KUKA KRL program: MyProgram_084().src

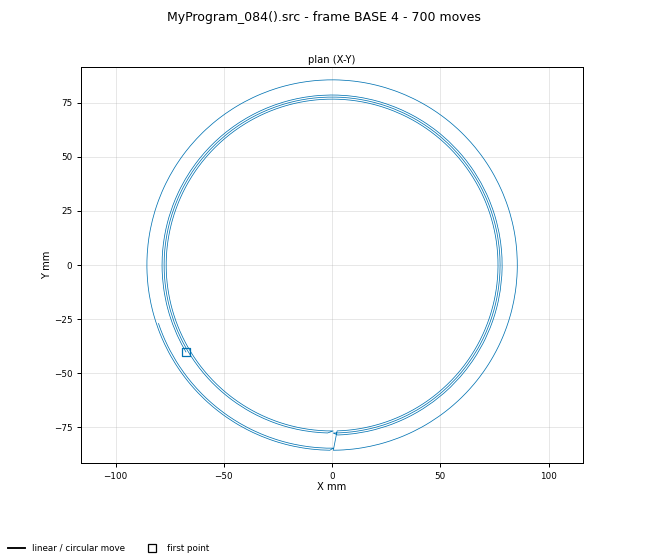
[picture p0: tool path of MyProgram_084().src in frame BASE 4, 700 of 700 moves have a stored position in this frame; points joined in program order, loops and branches not executed]
&ACCESS RVP
&REL 1
&PARAM TEMPLATE = C:\KRC\Roboter\Template\vorgabe
&PARAM EDITMASK = *
DEF MyProgram_084()
; ---- Setting reference (Base) ----
$BASE = BASE_DATA[4]

; --------------------------
; ---- Setting tool (TCP) ----
$TOOL = TOOL_DATA[3]
; --------------------------

$VEL.CP = VEL_APROX_PRINT
Startdeposition()
$VEL.CP = VEL_PRINT
LIN {X -67.4962,Y -40.1189,Z 83,A -155.1971,B 24.913,C -2.1538,E1 24.8612,E2 239.9035} C_DIS
LIN {X -69.3638,Y -36.7975,Z 83,A -157.7147,B 24.9119,C -2.1678,E1 24.8579,E2 242.401} C_DIS
LIN {X -71.5627,Y -32.3128,Z 83,A -161.7779,B 24.9119,C -2.1676,E1 24.853,E2 246.4869} C_DIS
LIN {X -73.6163,Y -27.3162,Z 83,A -165.4446,B 24.9104,C -2.1857,E1 24.8493,E2 250.1308} C_DIS
LIN {X -75.14,Y -22.7935,Z 83,A -168.9954,B 24.9097,C -2.1943,E1 24.8462,E2 253.6814} C_DIS
LIN {X -76.0413,Y -19.5719,Z 83,A -171.3695,B 24.9089,C -2.2034,E1 24.8445,E2 256.0476} C_DIS
LIN {X -76.5834,Y -17.3332,Z 83,A -173.4714,B 24.9094,C -2.1982,E1 24.8432,E2 258.1743} C_DIS
LIN {X -77.4433,Y -12.9563,Z 83,A -176.3604,B 24.9078,C -2.2172,E1 24.8417,E2 261.035} C_DIS
LIN {X -77.8334,Y -10.3623,Z 83,A -178.4896,B 24.9078,C -2.2179,E1 24.8409,E2 263.1752} C_DIS
LIN {X -78.3135,Y -5.7007,Z 83,A 178.2886,B 24.9064,C -2.2335,E1 24.8401,E2 266.3791} C_DIS
LIN {X -78.4754,Y -2.6451,Z 83,A 176.0932,B 24.9057,C -2.2415,E1 24.8398,E2 268.5686} C_DIS
LIN {X -78.5203,Y -0.1798,Z 83,A 174.0288,B 24.9058,C -2.2407,E1 24.8398,E2 270.6472} C_DIS
LIN {X -78.4321,Y 3.7214,Z 83,A 171.4381,B 24.9045,C -2.2561,E1 24.84,E2 273.217} C_DIS
LIN {X -78.2302,Y 6.7519,Z 83,A 169.0363,B 24.9043,C -2.2586,E1 24.8405,E2 275.6272} C_DIS
LIN {X -77.8931,Y 9.901,Z 83,A 166.9372,B 24.9032,C -2.2711,E1 24.8412,E2 277.7088} C_DIS
LIN {X -77.3929,Y 13.2579,Z 83,A 164.5258,B 24.9024,C -2.2806,E1 24.8423,E2 280.1121} C_DIS
LIN {X -76.7687,Y 16.4912,Z 83,A 161.8494,B 24.9024,C -2.2815,E1 24.8437,E2 282.8021} C_DIS
LIN {X -76.0396,Y 19.5784,Z 83,A 159.9359,B 24.9009,C -2.2986,E1 24.845,E2 284.6859} C_DIS
LIN {X -75.3479,Y 22.0927,Z 83,A 157.1821,B 24.9022,C -2.2837,E1 24.8471,E2 287.4912} C_DIS
LIN {X -73.5762,Y 27.4236,Z 83,A 153.3028,B 24.9006,C -2.3017,E1 24.8507,E2 291.3496} C_DIS
LIN {X -72.4018,Y 30.3864,Z 83,A 151.2241,B 24.8995,C -2.3147,E1 24.8529,E2 293.4087} C_DIS
LIN {X -70.9859,Y 33.5643,Z 83,A 148.6946,B 24.8988,C -2.3225,E1 24.8558,E2 295.9336} C_DIS
LIN {X -69.965,Y 35.6404,Z 83,A 146.6894,B 24.899,C -2.3197,E1 24.8583,E2 297.9562} C_DIS
LIN {X -67.7859,Y 39.6302,Z 83,A 143.1182,B 24.8988,C -2.323,E1 24.8633,E2 301.5383} C_DIS
LIN {X -65.3999,Y 43.4542,Z 83,A 139.7994,B 24.898,C -2.3314,E1 24.8683,E2 304.8537} C_DIS
LIN {X -63.0593,Y 46.7874,Z 83,A 137.4432,B 24.896,C -2.3546,E1 24.8721,E2 307.166} C_DIS
LIN {X -61.1985,Y 49.1953,Z 83,A 134.8431,B 24.8963,C -2.351,E1 24.8766,E2 309.7869} C_DIS
LIN {X -58.9466,Y 51.8721,Z 83,A 132.515,B 24.8952,C -2.3631,E1 24.8808,E2 312.0968} C_DIS
LIN {X -56.6359,Y 54.385,Z 83,A 129.9158,B 24.8949,C -2.3665,E1 24.8858,E2 314.6992} C_DIS
LIN {X -54.1507,Y 56.8608,Z 83,A 127.2895,B 24.8945,C -2.3708,E1 24.8911,E2 317.3261} C_DIS
LIN {X -51.3752,Y 59.3806,Z 83,A 124.709,B 24.8936,C -2.3809,E1 24.8964,E2 319.8928} C_DIS
LIN {X -48.7716,Y 61.536,Z 83,A 122.1128,B 24.8934,C -2.383,E1 24.9021,E2 322.4938} C_DIS
LIN {X -45.6856,Y 63.8605,Z 83,A 118.9561,B 24.8937,C -2.3802,E1 24.9092,E2 325.6683} C_DIS
LIN {X -42.8175,Y 65.8196,Z 83,A 115.9085,B 24.8944,C -2.372,E1 24.9164,E2 328.7453} C_DIS
LIN {X -39.3112,Y 67.9707,Z 83,A 113.6601,B 24.8922,C -2.3965,E1 24.9217,E2 330.9422} C_DIS
LIN {X -36.2205,Y 69.6677,Z 83,A 111.1741,B 24.8916,C -2.403,E1 24.9278,E2 333.4195} C_DIS
LIN {X -33.3372,Y 71.0916,Z 83,A 108.8468,B 24.8913,C -2.4072,E1 24.9336,E2 335.7429} C_DIS
LIN {X -30.2227,Y 72.4708,Z 83,A 105.584,B 24.8928,C -2.3906,E1 24.9422,E2 339.0527} C_DIS
LIN {X -26.6807,Y 73.848,Z 83,A 103.7974,B 24.8901,C -2.4199,E1 24.9467,E2 340.7734} C_DIS
LIN {X -22.5013,Y 75.2267,Z 83,A 100.3905,B 24.8902,C -2.4184,E1 24.9558,E2 344.1897} C_DIS
LIN {X -19.5528,Y 76.0462,Z 83,A 98.0831,B 24.8902,C -2.4187,E1 24.962,E2 346.5} C_DIS
LIN {X -16.2475,Y 76.8217,Z 83,A 95.2262,B 24.8909,C -2.4108,E1 24.9698,E2 349.3794} C_DIS
LIN {X -12.6748,Y 77.4904,Z 83,A 92.5015,B 24.8909,C -2.4108,E1 24.9773,E2 352.1066} C_DIS
LIN {X -8.3982,Y 78.0696,Z 83,A 89.8262,B 24.8896,C -2.4253,E1 24.9847,E2 354.7492} C_DIS
LIN {X -5.2916,Y 78.3411,Z 83,A 87.2441,B 24.8903,C -2.418,E1 24.9919,E2 357.3497} C_DIS
LIN {X -0.6851,Y 78.5169,Z 83,A 84.1569,B 24.8895,C -2.4265,E1 25.0005,E2 360.4172} C_DIS
LIN {X 2.6698,Y 78.4747,Z 83,A 81.8017,B 24.8892,C -2.4293,E1 25.007,E2 362.7652} C_DIS
LIN {X 7.1476,Y 78.1937,Z 83,A 78.4133,B 24.8895,C -2.4261,E1 25.0165,E2 366.1598} C_DIS
LIN {X 10.8186,Y 77.7711,Z 83,A 75.7639,B 24.8895,C -2.4268,E1 25.0238,E2 368.8054} C_DIS
LIN {X 14.4011,Y 77.189,Z 83,A 72.6133,B 24.8908,C -2.4119,E1 25.0326,E2 371.9879} C_DIS
LIN {X 18.7763,Y 76.2418,Z 83,A 69.7445,B 24.89,C -2.4213,E1 25.0403,E2 374.8305} C_DIS
LIN {X 21.894,Y 75.4069,Z 83,A 67.3804,B 24.8901,C -2.4194,E1 25.0466,E2 377.195} C_DIS
LIN {X 25.0356,Y 74.4215,Z 83,A 65.1631,B 24.8898,C -2.4228,E1 25.0525,E2 379.4002} C_DIS
LIN {X 29.0768,Y 72.9386,Z 83,A 62.2037,B 24.8896,C -2.4251,E1 25.0602,E2 382.348} C_DIS
LIN {X 32.2098,Y 71.6091,Z 83,A 59.24,B 24.8911,C -2.4086,E1 25.0679,E2 385.3435} C_DIS
LIN {X 35.5962,Y 69.9876,Z 83,A 56.777,B 24.8907,C -2.4132,E1 25.074,E2 387.7891} C_DIS
LIN {X 38.5611,Y 68.3994,Z 83,A 53.5616,B 24.893,C -2.3878,E1 25.082,E2 391.0551} C_DIS
LIN {X 41.7678,Y 66.4893,Z 83,A 51.5388,B 24.8915,C -2.404,E1 25.0867,E2 393.0331} C_DIS
LIN {X 43.7872,Y 65.1774,Z 83,A 49.4601,B 24.8926,C -2.3918,E1 25.0915,E2 395.1338} C_DIS
LIN {X 47.0859,Y 62.8352,Z 83,A 46.9103,B 24.892,C -2.3985,E1 25.0972,E2 397.6586} C_DIS
LIN {X 49.6786,Y 60.8068,Z 83,A 44.6975,B 24.892,C -2.3998,E1 25.102,E2 399.8603} C_DIS
LIN {X 53.8865,Y 57.1104,Z 83,A 40.3742,B 24.8933,C -2.3847,E1 25.1111,E2 404.202} C_DIS
LIN {X 58.1887,Y 52.722,Z 83,A 35.9551,B 24.894,C -2.3769,E1 25.1196,E2 408.6203} C_DIS
LIN {X 60.2405,Y 50.3634,Z 83,A 33.7323,B 24.8943,C -2.3735,E1 25.1237,E2 410.8412} C_DIS
LIN {X 62.2799,Y 47.818,Z 83,A 30.7906,B 24.8963,C -2.3509,E1 25.1288,E2 413.8223} C_DIS
LIN {X 64.1977,Y 45.2131,Z 83,A 28.9176,B 24.8955,C -2.3597,E1 25.1318,E2 415.6654} C_DIS
LIN {X 65.697,Y 43.0036,Z 83,A 26.6513,B 24.8968,C -2.3452,E1 25.1353,E2 417.9548} C_DIS
LIN {X 68.7357,Y 37.9588,Z 83,A 23.018,B 24.896,C -2.354,E1 25.1404,E2 421.5486} C_DIS
LIN {X 71.3889,Y 32.6985,Z 83,A 18.4593,B 24.8978,C -2.3341,E1 25.146,E2 426.1299} C_DIS
LIN {X 72.7,Y 29.6657,Z 83,A 15.8312,B 24.899,C -2.3206,E1 25.1489,E2 428.7754} C_DIS
LIN {X 74.1369,Y 25.8663,Z 83,A 13.2522,B 24.8987,C -2.3238,E1 25.1513,E2 431.3324} C_DIS
LIN {X 75.1174,Y 22.8665,Z 83,A 11.1082,B 24.8989,C -2.3218,E1 25.1531,E2 433.4689} C_DIS
LIN {X 75.9431,Y 19.954,Z 83,A 8.9268,B 24.8994,C -2.316,E1 25.1548,E2 435.6515} C_DIS
LIN {X 77.1297,Y 14.7088,Z 83,A 4.8617,B 24.9008,C -2.2996,E1 25.1572,E2 439.7318} C_DIS
LIN {X 77.7907,Y 10.6646,Z 83,A 1.7462,B 24.9019,C -2.2864,E1 25.1585,E2 442.8601} C_DIS
LIN {X 78.2253,Y 6.7842,Z 83,A -1.4293,B 24.9036,C -2.2673,E1 25.1594,E2 446.0619} C_DIS
LIN {X 78.4503,Y 3.3007,Z 83,A -4.5335,B 24.9057,C -2.2421,E1 25.1598,E2 449.2071} C_DIS
LIN {X 78.5112,Y -1.1833,Z 83,A -6.7555,B 24.9038,C -2.2641,E1 25.1598,E2 451.364} C_DIS
LIN {X 78.3698,Y -4.8681,Z 83,A -9.4916,B 24.9047,C -2.2541,E1 25.1594,E2 454.1076} C_DIS
LIN {X 77.6444,Y -11.6949,Z 83,A -14.1193,B 24.905,C -2.25,E1 25.1579,E2 458.7174} C_DIS
LIN {X 76.7025,Y -16.7949,Z 83,A -18.2468,B 24.9069,C -2.2273,E1 25.1558,E2 462.8745} C_DIS
LIN {X 76.0708,Y -19.4568,Z 83,A -20.7555,B 24.9088,C -2.2051,E1 25.154,E2 465.421} C_DIS
LIN {X 75.1954,Y -22.607,Z 83,A -22.6705,B 24.9082,C -2.2123,E1 25.1525,E2 467.3083} C_DIS
LIN {X 74.1573,Y -25.8085,Z 83,A -24.9152,B 24.9082,C -2.2112,E1 25.1505,E2 469.5427} C_DIS
LIN {X 73.0003,Y -28.9196,Z 83,A -27.6923,B 24.9098,C -2.1928,E1 25.1477,E2 472.3479} C_DIS
LIN {X 70.715,Y -34.1282,Z 83,A -31.553,B 24.9101,C -2.1894,E1 25.1433,E2 476.1958} C_DIS
LIN {X 69.6417,Y -36.2699,Z 83,A -33.8227,B 24.9118,C -2.1682,E1 25.1403,E2 478.5035} C_DIS
LIN {X 66.7563,Y -41.3403,Z 83,A -37.3323,B 24.9109,C -2.179,E1 25.1354,E2 481.9695} C_DIS
LIN {X 64.7944,Y -44.3529,Z 83,A -39.7414,B 24.9109,C -2.1783,E1 25.1317,E2 484.3682} C_DIS
LIN {X 62.0109,Y -48.1672,Z 83,A -43.4052,B 24.9123,C -2.1623,E1 25.1256,E2 488.0523} C_DIS
LIN {X 59.1059,Y -51.6897,Z 83,A -46.8855,B 24.9134,C -2.1491,E1 25.1193,E2 491.5478} C_DIS
LIN {X 54.589,Y -56.4393,Z 83,A -51.2634,B 24.9134,C -2.1497,E1 25.1109,E2 495.9053} C_DIS
LIN {X 51.7179,Y -59.0813,Z 83,A -54.4123,B 24.9146,C -2.134,E1 25.1043,E2 499.0789} C_DIS
LIN {X 46.8486,Y -63.0135,Z 83,A -59.0188,B 24.9155,C -2.1229,E1 25.0942,E2 503.6943} C_DIS
LIN {X 41.9662,Y -66.3653,Z 83,A -63.0379,B 24.9155,C -2.1235,E1 25.085,E2 507.6986} C_DIS
LIN {X 39.4629,Y -67.8835,Z 83,A -65.1401,B 24.9157,C -2.1206,E1 25.0799,E2 509.8011} C_DIS
LIN {X 36.5498,Y -69.4942,Z 83,A -68.3691,B 24.9179,C -2.0927,E1 25.0718,E2 513.087} C_DIS
LIN {X 33.6867,Y -70.9272,Z 83,A -70.1646,B 24.9169,C -2.1049,E1 25.0674,E2 514.8488} C_DIS
LIN {X 31.1101,Y -72.0942,Z 83,A -72.9633,B 24.9188,C -2.0803,E1 25.0601,E2 517.699} C_DIS
LIN {X 27.621,Y -73.5014,Z 83,A -74.9496,B 24.9174,C -2.0987,E1 25.055,E2 519.6373} C_DIS
LIN {X 24.8884,Y -74.4711,Z 83,A -76.8881,B 24.9172,C -2.1013,E1 25.0499,E2 521.566} C_DIS
LIN {X 19.7348,Y -75.9994,Z 83,A -81.0811,B 24.9182,C -2.089,E1 25.0386,E2 525.7809} C_DIS
LIN {X 16.2285,Y -76.8256,Z 83,A -83.6878,B 24.9182,C -2.0872,E1 25.0315,E2 528.3883} C_DIS
LIN {X 10.4449,Y -77.8227,Z 83,A -87.7619,B 24.9181,C -2.0901,E1 25.0203,E2 532.4516} C_DIS
LIN {X 5.4361,Y -78.3314,Z 83,A -91.4774,B 24.9183,C -2.087,E1 25.01,E2 536.1723} C_DIS
LIN {X 2.5825,Y -78.4774,Z 83,A -94.2573,B 24.9199,C -2.0666,E1 25.0021,E2 538.9997} C_DIS
LIN {X 2.5825,Y -78.4774,Z 83,A -94.2573,B 24.9199,C -2.0666,E1 25.0021,E2 538.9997} C_DIS
Enddeposition()
LIN {X 0.5144,Y -77.5659,Z 83,A -94.0454,B 24.9148,C -2.1314,E1 25.0031,E2 538.6341} C_DIS
Startdeposition()
$VEL.CP = VEL_PRINT
LIN {X 2.8882,Y -77.5153,Z 83,A -92.2446,B 24.9146,C -2.1333,E1 25.0082,E2 536.8292} C_DIS
LIN {X 5.9801,Y -77.3372,Z 83,A -90.1199,B 24.9149,C -2.1297,E1 25.014,E2 534.7141} C_DIS
LIN {X 9.4356,Y -76.9929,Z 83,A -87.6983,B 24.9151,C -2.127,E1 25.0207,E2 532.3005} C_DIS
LIN {X 11.649,Y -76.6884,Z 83,A -85.697,B 24.9142,C -2.1383,E1 25.0263,E2 530.2743} C_DIS
LIN {X 14.3793,Y -76.2239,Z 83,A -83.824,B 24.9145,C -2.1349,E1 25.0315,E2 528.4113} C_DIS
LIN {X 17.4499,Y -75.5795,Z 83,A -81.5326,B 24.9145,C -2.1363,E1 25.0377,E2 526.1198} C_DIS
LIN {X 20.4516,Y -74.8235,Z 83,A -78.6401,B 24.9128,C -2.1565,E1 25.0456,E2 523.184} C_DIS
LIN {X 23.5395,Y -73.9106,Z 83,A -77.1246,B 24.9146,C -2.1338,E1 25.0495,E2 521.725} C_DIS
LIN {X 25.6644,Y -73.199,Z 83,A -75.1482,B 24.9137,C -2.1453,E1 25.0548,E2 519.7251} C_DIS
LIN {X 29.4044,Y -71.7786,Z 83,A -72.2013,B 24.9134,C -2.1491,E1 25.0625,E2 516.7757} C_DIS
LIN {X 32.2204,Y -70.5603,Z 83,A -69.9294,B 24.9131,C -2.1527,E1 25.0683,E2 514.501} C_DIS
LIN {X 35.0376,Y -69.2041,Z 83,A -67.7153,B 24.9131,C -2.1536,E1 25.0738,E2 512.2906} C_DIS
LIN {X 39.2523,Y -66.9036,Z 83,A -64.4984,B 24.9133,C -2.1499,E1 25.0816,E2 509.0919} C_DIS
LIN {X 41.3924,Y -65.6015,Z 83,A -62.057,B 24.9116,C -2.1712,E1 25.0875,E2 506.608} C_DIS
LIN {X 43.7052,Y -64.0834,Z 83,A -60.217,B 24.9118,C -2.169,E1 25.0917,E2 504.7793} C_DIS
LIN {X 46.4318,Y -62.1361,Z 83,A -57.8094,B 24.9115,C -2.1721,E1 25.0972,E2 502.3729} C_DIS
LIN {X 49.6359,Y -59.6074,Z 83,A -55.1101,B 24.9118,C -2.1691,E1 25.103,E2 499.6909} C_DIS
LIN {X 51.4097,Y -58.0861,Z 83,A -52.9031,B 24.9102,C -2.1876,E1 25.1077,E2 497.4487} C_DIS
LIN {X 53.7596,Y -55.9167,Z 83,A -50.7486,B 24.9102,C -2.1868,E1 25.1121,E2 495.305} C_DIS
LIN {X 57.2392,Y -52.3493,Z 83,A -47.4138,B 24.9104,C -2.1852,E1 25.1185,E2 491.9883} C_DIS
LIN {X 58.6798,Y -50.7306,Z 83,A -45.3887,B 24.909,C -2.2023,E1 25.1223,E2 489.9319} C_DIS
LIN {X 60.3066,Y -48.784,Z 83,A -43.5847,B 24.9088,C -2.2051,E1 25.1255,E2 488.1297} C_DIS
LIN {X 62.3962,Y -46.0823,Z 83,A -40.7525,B 24.9074,C -2.2214,E1 25.1302,E2 485.2724} C_DIS
LIN {X 64.9028,Y -42.4789,Z 83,A -37.9102,B 24.9077,C -2.218,E1 25.1347,E2 482.4524} C_DIS
LIN {X 67.3301,Y -38.5154,Z 83,A -34.8501,B 24.9079,C -2.2162,E1 25.1391,E2 479.4122} C_DIS
LIN {X 68.3184,Y -36.7347,Z 83,A -32.9379,B 24.9064,C -2.2332,E1 25.1416,E2 477.4698} C_DIS
LIN {X 69.816,Y -33.8014,Z 83,A -30.5303,B 24.9059,C -2.2396,E1 25.1446,E2 475.0599} C_DIS
LIN {X 71.21,Y -30.7565,Z 83,A -27.5556,B 24.9039,C -2.2627,E1 25.148,E2 472.0469} C_DIS
LIN {X 72.7639,Y -26.8752,Z 83,A -25.0245,B 24.9046,C -2.2547,E1 25.1505,E2 469.5489} C_DIS
LIN {X 73.7569,Y -24.0147,Z 83,A -22.8028,B 24.9041,C -2.2611,E1 25.1525,E2 467.3244} C_DIS
LIN {X 74.7243,Y -20.8127,Z 83,A -20.498,B 24.9039,C -2.2636,E1 25.1543,E2 465.0269} C_DIS
LIN {X 75.4748,Y -17.903,Z 83,A -18.2233,B 24.9031,C -2.2723,E1 25.1558,E2 462.7448} C_DIS
LIN {X 76.0877,Y -15.0867,Z 83,A -15.6919,B 24.9015,C -2.2917,E1 25.1572,E2 460.1824} C_DIS
LIN {X 76.8338,Y -10.6486,Z 83,A -12.3703,B 24.9006,C -2.3022,E1 25.1586,E2 456.8556} C_DIS
LIN {X 77.2676,Y -6.8247,Z 83,A -9.8899,B 24.9008,C -2.2999,E1 25.1593,E2 454.3954} C_DIS
LIN {X 77.4854,Y -3.583,Z 83,A -7.5538,B 24.9003,C -2.3055,E1 25.1597,E2 452.0597} C_DIS
LIN {X 77.5685,Y 0.1521,Z 83,A -4.2817,B 24.8981,C -2.3304,E1 25.1597,E2 448.7484} C_DIS
LIN {X 77.4768,Y 3.7829,Z 83,A -2.0623,B 24.8986,C -2.3244,E1 25.1595,E2 446.5564} C_DIS
LIN {X 77.1234,Y 8.2944,Z 83,A 1.0166,B 24.8984,C -2.3267,E1 25.1587,E2 443.4904} C_DIS
LIN {X 76.4706,Y 13.0022,Z 83,A 4.4103,B 24.8978,C -2.334,E1 25.1574,E2 440.0994} C_DIS
LIN {X 76.0495,Y 15.2758,Z 83,A 7.1566,B 24.8944,C -2.3717,E1 25.1558,E2 437.2801} C_DIS
LIN {X 75.2014,Y 19.0159,Z 83,A 9.0938,B 24.8962,C -2.3523,E1 25.1546,E2 435.3999} C_DIS
LIN {X 74.4566,Y 21.7505,Z 83,A 11.3694,B 24.8951,C -2.3642,E1 25.1528,E2 433.1091} C_DIS
LIN {X 73.4182,Y 25.032,Z 83,A 13.8086,B 24.8947,C -2.3686,E1 25.1507,E2 430.6734} C_DIS
LIN {X 72.4124,Y 27.8089,Z 83,A 15.9437,B 24.8943,C -2.3735,E1 25.1486,E2 428.5387} C_DIS
LIN {X 71.2612,Y 30.639,Z 83,A 18.2781,B 24.8935,C -2.3823,E1 25.1461,E2 426.1962} C_DIS
LIN {X 69.2949,Y 34.8595,Z 83,A 21.6219,B 24.8929,C -2.3889,E1 25.1421,E2 422.8548} C_DIS
LIN {X 67.8522,Y 37.5887,Z 83,A 23.8874,B 24.8924,C -2.3946,E1 25.139,E2 420.5876} C_DIS
LIN {X 66.3667,Y 40.1528,Z 83,A 26.6002,B 24.8904,C -2.4165,E1 25.1351,E2 417.8371} C_DIS
LIN {X 64.3659,Y 43.288,Z 83,A 28.7997,B 24.8913,C -2.4067,E1 25.1318,E2 415.6718} C_DIS
LIN {X 62.4526,Y 46.0053,Z 83,A 30.9015,B 24.8917,C -2.402,E1 25.1284,E2 413.5911} C_DIS
LIN {X 60.212,Y 48.9007,Z 83,A 33.9636,B 24.8902,C -2.4193,E1 25.1231,E2 410.5026} C_DIS
LIN {X 58.0817,Y 51.4146,Z 83,A 36.4225,B 24.8896,C -2.4255,E1 25.1185,E2 408.04} C_DIS
LIN {X 55.3564,Y 54.3368,Z 83,A 39.217,B 24.8894,C -2.4272,E1 25.1132,E2 405.2536} C_DIS
LIN {X 53.3392,Y 56.3184,Z 83,A 41.3671,B 24.8889,C -2.4334,E1 25.1088,E2 403.098} C_DIS
LIN {X 50.0645,Y 59.2487,Z 83,A 44.5968,B 24.8883,C -2.4392,E1 25.1021,E2 399.8672} C_DIS
LIN {X 47.7466,Y 61.1328,Z 83,A 46.8891,B 24.8877,C -2.4458,E1 25.097,E2 397.5679} C_DIS
LIN {X 45.1584,Y 63.0674,Z 83,A 49.0892,B 24.8879,C -2.4444,E1 25.0921,E2 395.379} C_DIS
LIN {X 42.7881,Y 64.6989,Z 83,A 51.2522,B 24.8874,C -2.4489,E1 25.0871,E2 393.2125} C_DIS
LIN {X 39.8229,Y 66.5663,Z 83,A 53.6176,B 24.8877,C -2.4462,E1 25.0815,E2 390.8609} C_DIS
LIN {X 37.6936,Y 67.7936,Z 83,A 55.6054,B 24.887,C -2.4538,E1 25.0766,E2 388.8611} C_DIS
LIN {X 34.8797,Y 69.2848,Z 83,A 57.971,B 24.8867,C -2.4572,E1 25.0708,E2 386.494} C_DIS
LIN {X 32.6684,Y 70.353,Z 83,A 59.7698,B 24.8865,C -2.4589,E1 25.0662,E2 384.6957} C_DIS
LIN {X 28.6271,Y 72.0926,Z 83,A 63.0891,B 24.886,C -2.4643,E1 25.0577,E2 381.3715} C_DIS
LIN {X 25.9113,Y 73.1124,Z 83,A 65.2903,B 24.8857,C -2.4679,E1 25.0519,E2 379.1662} C_DIS
LIN {X 22.6551,Y 74.1864,Z 83,A 67.7318,B 24.8857,C -2.4673,E1 25.0454,E2 376.7308} C_DIS
LIN {X 19.7035,Y 75.0247,Z 83,A 70.0759,B 24.8854,C -2.471,E1 25.0391,E2 374.3817} C_DIS
LIN {X 16.7042,Y 75.748,Z 83,A 72.2866,B 24.8854,C -2.4702,E1 25.0331,E2 372.1758} C_DIS
LIN {X 13.3131,Y 76.418,Z 83,A 74.7891,B 24.8855,C -2.4698,E1 25.0262,E2 369.6772} C_DIS
LIN {X 10.7478,Y 76.8198,Z 83,A 76.6732,B 24.8855,C -2.4694,E1 25.021,E2 367.7958} C_DIS
LIN {X 7.8323,Y 77.1717,Z 83,A 79.0416,B 24.885,C -2.4753,E1 25.0144,E2 365.4151} C_DIS
LIN {X 4.3652,Y 77.4449,Z 83,A 81.3855,B 24.8856,C -2.4691,E1 25.0079,E2 363.0869} C_DIS
LIN {X 1.7743,Y 77.5483,Z 83,A 83.5183,B 24.885,C -2.4749,E1 25.0019,E2 360.9407} C_DIS
LIN {X -1.6494,Y 77.5506,Z 83,A 86.1229,B 24.8849,C -2.4764,E1 24.9946,E2 358.3325} C_DIS
LIN {X -5.5687,Y 77.3684,Z 83,A 88.8303,B 24.8855,C -2.47,E1 24.9871,E2 355.6393} C_DIS
LIN {X -8.6281,Y 77.0875,Z 83,A 91.0546,B 24.8857,C -2.4676,E1 24.981,E2 353.4195} C_DIS
LIN {X -11.2785,Y 76.7444,Z 83,A 93.139,B 24.8855,C -2.4694,E1 24.9752,E2 351.3293} C_DIS
LIN {X -14.1625,Y 76.2652,Z 83,A 95.2643,B 24.8858,C -2.4668,E1 24.9694,E2 349.2079} C_DIS
LIN {X -17.0711,Y 75.667,Z 83,A 97.4153,B 24.8861,C -2.4638,E1 24.9635,E2 347.0614} C_DIS
LIN {X -19.9888,Y 74.9485,Z 83,A 99.6427,B 24.8862,C -2.4619,E1 24.9575,E2 344.8355} C_DIS
LIN {X -22.8094,Y 74.1385,Z 83,A 101.7457,B 24.8866,C -2.4578,E1 24.9519,E2 342.7386} C_DIS
LIN {X -26.1046,Y 73.0446,Z 83,A 104.7355,B 24.8859,C -2.4659,E1 24.9439,E2 339.7238} C_DIS
LIN {X -29.7731,Y 71.6273,Z 83,A 107.33,B 24.887,C -2.4537,E1 24.9372,E2 337.1525} C_DIS
LIN {X -32.6232,Y 70.3741,Z 83,A 109.5483,B 24.8875,C -2.4482,E1 24.9316,E2 334.942} C_DIS
LIN {X -35.3138,Y 69.063,Z 83,A 111.7377,B 24.8879,C -2.4441,E1 24.9262,E2 332.7565} C_DIS
LIN {X -37.9124,Y 67.6714,Z 83,A 114.0762,B 24.8879,C -2.4446,E1 24.9204,E2 330.4102} C_DIS
LIN {X -41.1307,Y 65.765,Z 83,A 116.6178,B 24.8888,C -2.4339,E1 24.9144,E2 327.8863} C_DIS
LIN {X -43.3064,Y 64.3534,Z 83,A 118.7539,B 24.8886,C -2.4359,E1 24.9094,E2 325.7385} C_DIS
LIN {X -45.9969,Y 62.4588,Z 83,A 121.2927,B 24.8888,C -2.4337,E1 24.9036,E2 323.1959} C_DIS
LIN {X -48.8491,Y 60.2539,Z 83,A 124.2101,B 24.8888,C -2.4346,E1 24.8972,E2 320.2657} C_DIS
LIN {X -53.1426,Y 56.5029,Z 83,A 128.2975,B 24.8899,C -2.4218,E1 24.8888,E2 316.1923} C_DIS
LIN {X -56.3746,Y 53.278,Z 83,A 131.9463,B 24.89,C -2.4207,E1 24.8817,E2 312.5306} C_DIS
LIN {X -60.1136,Y 49.0222,Z 83,A 135.9277,B 24.8915,C -2.4048,E1 24.8745,E2 308.5688} C_DIS
LIN {X -62.5421,Y 45.883,Z 83,A 139.1292,B 24.8915,C -2.4038,E1 24.8691,E2 305.3543} C_DIS
LIN {X -64.4973,Y 43.094,Z 83,A 141.2888,B 24.893,C -2.3879,E1 24.8658,E2 303.2219} C_DIS
LIN {X -66.3315,Y 40.2107,Z 83,A 143.6789,B 24.8939,C -2.3775,E1 24.8623,E2 300.8444} C_DIS
LIN {X -68.4577,Y 36.4746,Z 83,A 146.7832,B 24.8949,C -2.3666,E1 24.8581,E2 297.7499} C_DIS
LIN {X -69.6089,Y 34.2262,Z 83,A 148.8571,B 24.8949,C -2.3663,E1 24.8555,E2 295.6656} C_DIS
LIN {X -71.0502,Y 31.1231,Z 83,A 151.2823,B 24.8958,C -2.3562,E1 24.8527,E2 293.2511} C_DIS
LIN {X -72.5609,Y 27.4168,Z 83,A 154.1505,B 24.8968,C -2.3451,E1 24.8498,E2 290.3934} C_DIS
LIN {X -73.82,Y 23.8197,Z 83,A 157.491,B 24.8964,C -2.3494,E1 24.8468,E2 287.0236} C_DIS
LIN {X -74.8558,Y 20.3319,Z 83,A 159.8661,B 24.8978,C -2.3333,E1 24.845,E2 284.6733} C_DIS
LIN {X -75.6393,Y 17.191,Z 83,A 162.2116,B 24.8986,C -2.3247,E1 24.8435,E2 282.3346} C_DIS
LIN {X -76.2063,Y 14.4705,Z 83,A 164.1579,B 24.8994,C -2.3156,E1 24.8424,E2 280.3985} C_DIS
LIN {X -76.6093,Y 12.1603,Z 83,A 165.84,B 24.9,C -2.3089,E1 24.8416,E2 278.7225} C_DIS
LIN {X -76.9542,Y 9.7401,Z 83,A 167.8187,B 24.9001,C -2.3074,E1 24.8409,E2 276.7355} C_DIS
LIN {X -77.2825,Y 6.6628,Z 83,A 170.2377,B 24.9005,C -2.3033,E1 24.8402,E2 274.3117} C_DIS
LIN {X -77.4857,Y 3.5753,Z 83,A 172.4935,B 24.9012,C -2.2953,E1 24.8399,E2 272.0614} C_DIS
LIN {X -77.5664,Y 0.5388,Z 83,A 174.7982,B 24.9016,C -2.2897,E1 24.8398,E2 269.7563} C_DIS
LIN {X -77.5236,Y -2.631,Z 83,A 177.1476,B 24.9023,C -2.2824,E1 24.8399,E2 267.4101} C_DIS
LIN {X -77.3599,Y -5.6866,Z 83,A 179.3144,B 24.9031,C -2.273,E1 24.8403,E2 265.2528} C_DIS
LIN {X -77.1118,Y -8.4048,Z 83,A -178.7655,B 24.9038,C -2.2643,E1 24.8409,E2 263.3419} C_DIS
LIN {X -76.7318,Y -11.3672,Z 83,A -176.3396,B 24.9039,C -2.2628,E1 24.8418,E2 260.9051} C_DIS
LIN {X -76.2488,Y -14.2499,Z 83,A -174.1416,B 24.9044,C -2.2571,E1 24.8429,E2 258.7077} C_DIS
LIN {X -75.5667,Y -17.5055,Z 83,A -171.6417,B 24.905,C -2.2507,E1 24.8444,E2 256.2085} C_DIS
LIN {X -74.6882,Y -20.94,Z 83,A -169.0819,B 24.9058,C -2.2413,E1 24.8462,E2 253.6562} C_DIS
LIN {X -72.9011,Y -26.4991,Z 83,A -165.0069,B 24.9073,C -2.2226,E1 24.8498,E2 249.6024} C_DIS
LIN {X -71.3698,Y -30.3842,Z 83,A -161.1864,B 24.9065,C -2.2321,E1 24.8538,E2 245.7379} C_DIS
LIN {X -69.5568,Y -34.3311,Z 83,A -158.7383,B 24.9089,C -2.2041,E1 24.8567,E2 243.3433} C_DIS
LIN {X -68.6533,Y -36.1038,Z 83,A -156.9925,B 24.9086,C -2.2071,E1 24.859,E2 241.5813} C_DIS
LIN {X -67.2464,Y -38.6612,Z 83,A -154.2667,B 24.9079,C -2.2157,E1 24.8628,E2 238.8205} C_DIS
LIN {X -65.462,Y -41.6126,Z 83,A -151.5496,B 24.9081,C -2.2135,E1 24.8669,E2 236.0949} C_DIS
LIN {X -63.5981,Y -44.408,Z 83,A -149.2472,B 24.909,C -2.2027,E1 24.8705,E2 233.8069} C_DIS
LIN {X -61.2909,Y -47.542,Z 83,A -146.8133,B 24.9105,C -2.1845,E1 24.8745,E2 231.4048} C_DIS
LIN {X -59.4137,Y -49.869,Z 83,A -144.4279,B 24.9105,C -2.184,E1 24.8788,E2 229.0097} C_DIS
LIN {X -57.4191,Y -52.1533,Z 83,A -142.329,B 24.9112,C -2.1753,E1 24.8827,E2 226.9221} C_DIS
LIN {X -55.4672,Y -54.2247,Z 83,A -140.195,B 24.9115,C -2.1717,E1 24.8868,E2 224.7875} C_DIS
LIN {X -53.0598,Y -56.5812,Z 83,A -138.0202,B 24.9126,C -2.1585,E1 24.8912,E2 222.6351} C_DIS
LIN {X -51.3842,Y -58.1089,Z 83,A -135.9636,B 24.9121,C -2.1651,E1 24.8955,E2 220.5547} C_DIS
LIN {X -48.9908,Y -60.139,Z 83,A -133.7365,B 24.9126,C -2.1584,E1 24.9002,E2 218.3349} C_DIS
LIN {X -46.6223,Y -61.993,Z 83,A -131.4124,B 24.9127,C -2.1572,E1 24.9054,E2 216.0053} C_DIS
LIN {X -43.967,Y -63.9042,Z 83,A -128.6946,B 24.9124,C -2.1612,E1 24.9117,E2 213.2687} C_DIS
LIN {X -39.599,Y -66.6986,Z 83,A -125.3193,B 24.9138,C -2.1434,E1 24.9196,E2 209.9252} C_DIS
LIN {X -37.2139,Y -68.0585,Z 83,A -123.2755,B 24.914,C -2.141,E1 24.9246,E2 207.881} C_DIS
LIN {X -34.861,Y -69.2938,Z 83,A -121.196,B 24.914,C -2.1417,E1 24.9298,E2 205.7943} C_DIS
LIN {X -31.4541,Y -70.9056,Z 83,A -118.4135,B 24.9142,C -2.1385,E1 24.9368,E2 203.0124} C_DIS
LIN {X -27.675,Y -72.4631,Z 83,A -115.6782,B 24.9151,C -2.1279,E1 24.9439,E2 200.2964} C_DIS
LIN {X -25.38,Y -73.2989,Z 83,A -113.5956,B 24.9146,C -2.1339,E1 24.9494,E2 198.1954} C_DIS
LIN {X -22.461,Y -74.2458,Z 83,A -111.28,B 24.9146,C -2.1336,E1 24.9556,E2 195.8765} C_DIS
LIN {X -19.5292,Y -75.0695,Z 83,A -109.0211,B 24.9147,C -2.1325,E1 24.9617,E2 193.6167} C_DIS
LIN {X -16.1653,Y -75.8656,Z 83,A -106.5455,B 24.915,C -2.1291,E1 24.9684,E2 191.146} C_DIS
LIN {X -13.2264,Y -76.4331,Z 83,A -104.1817,B 24.9147,C -2.1326,E1 24.9749,E2 188.7715} C_DIS
LIN {X -9.0429,Y -77.0389,Z 83,A -100.8733,B 24.9143,C -2.1372,E1 24.9841,E2 185.4496} C_DIS
LIN {X -5.0773,Y -77.4016,Z 83,A -98.2255,B 24.915,C -2.1289,E1 24.9914,E2 182.8205} C_DIS
LIN {X -2.1127,Y -77.5395,Z 83,A -95.6562,B 24.9141,C -2.1399,E1 24.9987,E2 180.2247} C_DIS
LIN {X -2.1127,Y -77.5395,Z 83,A -95.6562,B 24.9141,C -2.1399,E1 24.9987,E2 180.2247} C_DIS
Enddeposition()
LIN {X 0.5155,Y -76.6129,Z 83,A -95.085,B 24.9158,C -2.1184,E1 25.0001,E2 179.7046} C_DIS
Startdeposition()
$VEL.CP = VEL_PRINT
LIN {X -2.6348,Y -76.5712,Z 83,A -97.4897,B 24.916,C -2.1166,E1 24.9934,E2 182.1137} C_DIS
LIN {X -5.4381,Y -76.4232,Z 83,A -99.4687,B 24.9157,C -2.1198,E1 24.9879,E2 184.0856} C_DIS
LIN {X -8.2769,Y -76.1681,Z 83,A -101.725,B 24.916,C -2.1166,E1 24.9816,E2 186.3509} C_DIS
LIN {X -11.2602,Y -75.7853,Z 83,A -104.11,B 24.9162,C -2.1134,E1 24.975,E2 188.7453} C_DIS
LIN {X -14.0308,Y -75.3217,Z 83,A -106.0437,B 24.9158,C -2.1186,E1 24.9697,E2 190.6687} C_DIS
LIN {X -16.0658,Y -74.9131,Z 83,A -107.6696,B 24.9159,C -2.1173,E1 24.9652,E2 192.2996} C_DIS
LIN {X -18.8183,Y -74.2694,Z 83,A -109.5982,B 24.9154,C -2.1233,E1 24.96,E2 194.2164} C_DIS
LIN {X -21.2511,Y -73.6107,Z 83,A -111.6784,B 24.9158,C -2.1193,E1 24.9544,E2 196.3094} C_DIS
LIN {X -24.0364,Y -72.7494,Z 83,A -113.6696,B 24.9152,C -2.1259,E1 24.9491,E2 198.2884} C_DIS
LIN {X -26.0023,Y -72.0691,Z 83,A -115.2287,B 24.9152,C -2.1272,E1 24.945,E2 199.8477} C_DIS
LIN {X -29.3612,Y -70.768,Z 83,A -118.2139,B 24.9155,C -2.1221,E1 24.9372,E2 202.8514} C_DIS
LIN {X -32.1105,Y -69.5628,Z 83,A -120.3607,B 24.9151,C -2.1272,E1 24.9318,E2 204.9915} C_DIS
LIN {X -34.6404,Y -68.3382,Z 83,A -122.4711,B 24.915,C -2.1295,E1 24.9265,E2 207.102} C_DIS
LIN {X -36.9479,Y -67.1198,Z 83,A -124.3599,B 24.9146,C -2.1336,E1 24.9219,E2 208.9861} C_DIS
LIN {X -39.2855,Y -65.7782,Z 83,A -126.3373,B 24.9143,C -2.1375,E1 24.9171,E2 210.9604} C_DIS
LIN {X -41.2172,Y -64.5847,Z 83,A -128.1854,B 24.9144,C -2.1362,E1 24.9127,E2 212.8174} C_DIS
LIN {X -43.5999,Y -63.0006,Z 83,A -130.3037,B 24.9141,C -2.1402,E1 24.9078,E2 214.9333} C_DIS
LIN {X -46.2384,Y -61.0908,Z 83,A -132.8157,B 24.9139,C -2.1424,E1 24.9022,E2 217.4489} C_DIS
LIN {X -48.6089,Y -59.2233,Z 83,A -135.0777,B 24.9136,C -2.1463,E1 24.8973,E2 219.7099} C_DIS
LIN {X -50.8275,Y -57.3298,Z 83,A -137.2164,B 24.9132,C -2.1516,E1 24.8928,E2 221.8445} C_DIS
LIN {X -53.1014,Y -55.229,Z 83,A -139.5545,B 24.9128,C -2.1557,E1 24.888,E2 224.1824} C_DIS
LIN {X -55.2347,Y -53.0956,Z 83,A -141.8711,B 24.9126,C -2.159,E1 24.8835,E2 226.501} C_DIS
LIN {X -57.3922,Y -50.7578,Z 83,A -144.0024,B 24.9116,C -2.1704,E1 24.8795,E2 228.6147} C_DIS
LIN {X -58.9923,Y -48.8868,Z 83,A -145.9876,B 24.9116,C -2.171,E1 24.8759,E2 230.6074} C_DIS
LIN {X -60.7404,Y -46.697,Z 83,A -148.0801,B 24.9112,C -2.1761,E1 24.8723,E2 232.6977} C_DIS
LIN {X -62.2422,Y -44.6762,Z 83,A -150.0752,B 24.911,C -2.1779,E1 24.869,E2 234.6982} C_DIS
LIN {X -63.8267,Y -42.3819,Z 83,A -152.1717,B 24.9106,C -2.1829,E1 24.8658,E2 236.7933} C_DIS
LIN {X -65.5213,Y -39.7111,Z 83,A -154.4127,B 24.9099,C -2.192,E1 24.8625,E2 239.0239} C_DIS
LIN {X -66.7665,Y -37.5806,Z 83,A -156.185,B 24.9093,C -2.1987,E1 24.86,E2 240.7895} C_DIS
LIN {X -67.6895,Y -35.8913,Z 83,A -157.8383,B 24.9094,C -2.1974,E1 24.8578,E2 242.4547} C_DIS
LIN {X -68.9861,Y -33.3308,Z 83,A -160.0125,B 24.909,C -2.2026,E1 24.8551,E2 244.6281} C_DIS
LIN {X -70.3562,Y -30.3332,Z 83,A -162.3104,B 24.9081,C -2.2136,E1 24.8525,E2 246.9124} C_DIS
LIN {X -71.2202,Y -28.2444,Z 83,A -164.1976,B 24.9081,C -2.2136,E1 24.8505,E2 248.8099} C_DIS
LIN {X -72.2027,Y -25.6292,Z 83,A -166.3083,B 24.9076,C -2.2193,E1 24.8485,E2 250.9193} C_DIS
LIN {X -73.088,Y -22.9834,Z 83,A -168.3877,B 24.9071,C -2.2256,E1 24.8467,E2 252.9955} C_DIS
LIN {X -73.8413,Y -20.4374,Z 83,A -170.1784,B 24.9062,C -2.2362,E1 24.8454,E2 254.7712} C_DIS
LIN {X -74.3682,Y -18.4241,Z 83,A -171.838,B 24.906,C -2.2384,E1 24.8442,E2 256.4351} C_DIS
LIN {X -74.9581,Y -15.8584,Z 83,A -173.8431,B 24.9056,C -2.2436,E1 24.843,E2 258.4398} C_DIS
LIN {X -75.4541,Y -13.2951,Z 83,A -175.719,B 24.9049,C -2.2515,E1 24.8421,E2 260.3079} C_DIS
LIN {X -75.8164,Y -11.0429,Z 83,A -177.6002,B 24.9049,C -2.2526,E1 24.8413,E2 262.1977} C_DIS
LIN {X -76.1732,Y -8.2283,Z 83,A -179.547,B 24.9039,C -2.2634,E1 24.8406,E2 264.1303} C_DIS
LIN {X -76.3943,Y -5.8306,Z 83,A 178.6108,B 24.9035,C -2.2681,E1 24.8402,E2 265.9724} C_DIS
LIN {X -76.5339,Y -3.554,Z 83,A 176.9216,B 24.903,C -2.2739,E1 24.8399,E2 267.6579} C_DIS
LIN {X -76.6078,Y -1.1467,Z 83,A 175.0823,B 24.9026,C -2.2787,E1 24.8398,E2 269.4968} C_DIS
LIN {X -76.6017,Y 1.4788,Z 83,A 173.0389,B 24.9022,C -2.283,E1 24.8398,E2 271.5422} C_DIS
LIN {X -76.5136,Y 3.9675,Z 83,A 171.066,B 24.9019,C -2.2863,E1 24.8401,E2 273.519} C_DIS
LIN {X -76.3349,Y 6.5736,Z 83,A 169.2854,B 24.901,C -2.2966,E1 24.8405,E2 275.2857} C_DIS
LIN {X -76.1274,Y 8.6427,Z 83,A 167.7202,B 24.9006,C -2.3014,E1 24.8409,E2 276.849} C_DIS
LIN {X -75.8179,Y 11.0322,Z 83,A 165.8781,B 24.9002,C -2.3061,E1 24.8416,E2 278.6907} C_DIS
LIN {X -75.4538,Y 13.2966,Z 83,A 163.9856,B 24.9002,C -2.3074,E1 24.8425,E2 280.5914} C_DIS
LIN {X -74.9121,Y 16.0702,Z 83,A 161.861,B 24.8996,C -2.3138,E1 24.8437,E2 282.7133} C_DIS
LIN {X -74.2711,Y 18.8116,Z 83,A 159.9292,B 24.8986,C -2.3245,E1 24.8449,E2 284.6308} C_DIS
LIN {X -73.7476,Y 20.7678,Z 83,A 158.1938,B 24.8986,C -2.324,E1 24.8462,E2 286.3775} C_DIS
LIN {X -72.9599,Y 23.386,Z 83,A 156.1268,B 24.8982,C -2.3298,E1 24.848,E2 288.4426} C_DIS
LIN {X -71.9478,Y 26.3349,Z 83,A 153.7448,B 24.8976,C -2.3357,E1 24.8502,E2 290.8238} C_DIS
LIN {X -70.7813,Y 29.3295,Z 83,A 151.4607,B 24.8967,C -2.3458,E1 24.8525,E2 293.0966} C_DIS
LIN {X -69.9585,Y 31.239,Z 83,A 150.0121,B 24.8961,C -2.353,E1 24.8541,E2 294.536} C_DIS
LIN {X -68.9416,Y 33.4234,Z 83,A 148.0543,B 24.896,C -2.3546,E1 24.8565,E2 296.5006} C_DIS
LIN {X -67.6486,Y 35.969,Z 83,A 146.0113,B 24.8952,C -2.363,E1 24.8591,E2 298.5345} C_DIS
LIN {X -66.5515,Y 37.9599,Z 83,A 144.1102,B 24.8952,C -2.3631,E1 24.8617,E2 300.4453} C_DIS
LIN {X -64.8343,Y 40.824,Z 83,A 141.7979,B 24.8942,C -2.3746,E1 24.8651,E2 302.7421} C_DIS
LIN {X -63.3195,Y 43.1357,Z 83,A 139.618,B 24.8939,C -2.3776,E1 24.8684,E2 304.9258} C_DIS
LIN {X -61.9112,Y 45.1335,Z 83,A 137.6882,B 24.8937,C -2.38,E1 24.8716,E2 306.859} C_DIS
LIN {X -60.085,Y 47.5373,Z 83,A 135.5212,B 24.893,C -2.3882,E1 24.8753,E2 309.017} C_DIS
LIN {X -58.1746,Y 49.8574,Z 83,A 133.112,B 24.8928,C -2.39,E1 24.8796,E2 311.4328} C_DIS
LIN {X -55.9852,Y 52.3041,Z 83,A 130.7305,B 24.8921,C -2.3979,E1 24.8841,E2 313.806} C_DIS
LIN {X -54.0446,Y 54.3071,Z 83,A 128.6373,B 24.8917,C -2.4027,E1 24.8882,E2 315.8966} C_DIS
LIN {X -51.8547,Y 56.4012,Z 83,A 126.3819,B 24.8912,C -2.4082,E1 24.8928,E2 318.1481} C_DIS
LIN {X -49.5633,Y 58.4252,Z 83,A 123.9716,B 24.891,C -2.4103,E1 24.8979,E2 320.5629} C_DIS
LIN {X -47.1092,Y 60.4228,Z 83,A 121.7429,B 24.8902,C -2.4187,E1 24.9027,E2 322.7798} C_DIS
LIN {X -44.8675,Y 62.1057,Z 83,A 119.4628,B 24.8902,C -2.4185,E1 24.9078,E2 325.0687} C_DIS
LIN {X -42.3945,Y 63.8183,Z 83,A 117.3014,B 24.8896,C -2.425,E1 24.9128,E2 327.2216} C_DIS
LIN {X -40.002,Y 65.3445,Z 83,A 115.3586,B 24.8889,C -2.4335,E1 24.9174,E2 329.1505} C_DIS
LIN {X -37.9302,Y 66.5686,Z 83,A 113.4044,B 24.8889,C -2.4328,E1 24.9221,E2 331.1122} C_DIS
LIN {X -35.9317,Y 67.6682,Z 83,A 111.625,B 24.8889,C -2.4338,E1 24.9265,E2 332.8942} C_DIS
LIN {X -33.4224,Y 68.9421,Z 83,A 109.5376,B 24.8885,C -2.4375,E1 24.9317,E2 334.9781} C_DIS
LIN {X -31.0538,Y 70.042,Z 83,A 107.6517,B 24.8881,C -2.4421,E1 24.9365,E2 336.8577} C_DIS
LIN {X -28.6487,Y 71.0586,Z 83,A 105.78,B 24.8876,C -2.4469,E1 24.9413,E2 338.7222} C_DIS
LIN {X -26.0268,Y 72.0602,Z 83,A 103.657,B 24.8874,C -2.449,E1 24.9469,E2 340.8446} C_DIS
LIN {X -23.3179,Y 72.9819,Z 83,A 101.5257,B 24.8872,C -2.4518,E1 24.9525,E2 342.9733} C_DIS
LIN {X -21.3301,Y 73.5883,Z 83,A 99.9995,B 24.887,C -2.4542,E1 24.9566,E2 344.4963} C_DIS
LIN {X -19.454,Y 74.106,Z 83,A 98.4648,B 24.887,C -2.4536,E1 24.9607,E2 346.0346} C_DIS
LIN {X -17.5043,Y 74.59,Z 83,A 96.8464,B 24.8872,C -2.452,E1 24.9651,E2 347.659} C_DIS
LIN {X -14.7398,Y 75.1851,Z 83,A 94.7004,B 24.8871,C -2.453,E1 24.971,E2 349.8054} C_DIS
LIN {X -12.1548,Y 75.647,Z 83,A 92.8336,B 24.8867,C -2.4569,E1 24.9761,E2 351.6646} C_DIS
LIN {X -9.5706,Y 76.0163,Z 83,A 90.8488,B 24.8867,C -2.4573,E1 24.9816,E2 353.6501} C_DIS
LIN {X -7.3037,Y 76.2675,Z 83,A 89.0989,B 24.8867,C -2.457,E1 24.9865,E2 355.4016} C_DIS
LIN {X -4.667,Y 76.4749,Z 83,A 87.1942,B 24.8864,C -2.4597,E1 24.9918,E2 357.3006} C_DIS
LIN {X -1.8615,Y 76.5947,Z 83,A 85.0905,B 24.8864,C -2.4603,E1 24.9976,E2 359.4032} C_DIS
LIN {X 0.7464,Y 76.6128,Z 83,A 83.2255,B 24.8861,C -2.4629,E1 25.0028,E2 361.2619} C_DIS
LIN {X 2.8223,Y 76.5654,Z 83,A 81.4492,B 24.8867,C -2.4571,E1 25.0078,E2 363.0516} C_DIS
LIN {X 5.8645,Y 76.3915,Z 83,A 79.1944,B 24.8867,C -2.4577,E1 25.0141,E2 365.304} C_DIS
LIN {X 8.661,Y 76.1252,Z 83,A 77.3219,B 24.8861,C -2.4636,E1 25.0193,E2 367.1613} C_DIS
LIN {X 11.0469,Y 75.8158,Z 83,A 75.2844,B 24.8867,C -2.4567,E1 25.0249,E2 369.2134} C_DIS
LIN {X 14.0201,Y 75.3237,Z 83,A 73.1561,B 24.8865,C -2.4593,E1 25.0308,E2 371.3333} C_DIS
LIN {X 16.0714,Y 74.9118,Z 83,A 71.5211,B 24.8867,C -2.4567,E1 25.0352,E2 372.9725} C_DIS
LIN {X 18.8201,Y 74.2689,Z 83,A 69.5989,B 24.8864,C -2.4607,E1 25.0404,E2 374.8824} C_DIS
LIN {X 20.6342,Y 73.7855,Z 83,A 68.1968,B 24.8864,C -2.4598,E1 25.0442,E2 376.2843} C_DIS
LIN {X 22.9452,Y 73.0999,Z 83,A 66.2546,B 24.8869,C -2.4546,E1 25.0494,E2 378.2353} C_DIS
LIN {X 25.6162,Y 72.2072,Z 83,A 64.1537,B 24.8871,C -2.453,E1 25.055,E2 380.336} C_DIS
LIN {X 28.2921,Y 71.2015,Z 83,A 62.1246,B 24.887,C -2.454,E1 25.0602,E2 382.3584} C_DIS
LIN {X 30.3933,Y 70.33,Z 83,A 60.4657,B 24.887,C -2.4533,E1 25.0645,E2 384.0148} C_DIS
LIN {X 32.1032,Y 69.5661,Z 83,A 58.8842,B 24.8877,C -2.4467,E1 25.0685,E2 385.6082} C_DIS
LIN {X 34.6329,Y 68.342,Z 83,A 56.7856,B 24.8879,C -2.4442,E1 25.0738,E2 387.707} C_DIS
LIN {X 36.9397,Y 67.1244,Z 83,A 54.9126,B 24.8879,C -2.4437,E1 25.0784,E2 389.5757} C_DIS
LIN {X 39.3765,Y 65.7244,Z 83,A 52.9306,B 24.8879,C -2.4441,E1 25.0832,E2 391.5508} C_DIS
LIN {X 41.5824,Y 64.3503,Z 83,A 50.835,B 24.8886,C -2.4368,E1 25.0881,E2 393.6569} C_DIS
LIN {X 43.5233,Y 63.0538,Z 83,A 49.0719,B 24.8889,C -2.4335,E1 25.0922,E2 395.422} C_DIS
LIN {X 45.6471,Y 61.5351,Z 83,A 47.0632,B 24.8893,C -2.4285,E1 25.0967,E2 397.4354} C_DIS
LIN {X 47.9548,Y 59.7535,Z 83,A 44.9734,B 24.8894,C -2.4271,E1 25.1013,E2 399.5206} C_DIS
LIN {X 50.1336,Y 57.9374,Z 83,A 42.8352,B 24.8899,C -2.4226,E1 25.1059,E2 401.6612} C_DIS
LIN {X 52.2246,Y 56.06,Z 83,A 40.7403,B 24.8902,C -2.4186,E1 25.1102,E2 403.7571} C_DIS
LIN {X 54.2458,Y 54.1067,Z 83,A 38.6404,B 24.8906,C -2.4143,E1 25.1144,E2 405.8585} C_DIS
LIN {X 56.388,Y 51.8691,Z 83,A 36.3844,B 24.8909,C -2.411,E1 25.1187,E2 408.1123} C_DIS
LIN {X 58.3864,Y 49.6089,Z 83,A 34.0338,B 24.8916,C -2.4031,E1 25.123,E2 410.471} C_DIS
LIN {X 60.3965,Y 47.1431,Z 83,A 31.8112,B 24.8917,C -2.4021,E1 25.1269,E2 412.6857} C_DIS
LIN {X 62.0865,Y 44.8941,Z 83,A 29.8305,B 24.8919,C -2.4006,E1 25.1301,E2 414.6604} C_DIS
LIN {X 63.4773,Y 42.9027,Z 83,A 27.9196,B 24.8925,C -2.3932,E1 25.1332,E2 416.5793} C_DIS
LIN {X 64.8508,Y 40.7974,Z 83,A 25.932,B 24.8932,C -2.3852,E1 25.1362,E2 418.5759} C_DIS
LIN {X 66.5657,Y 37.9353,Z 83,A 23.5341,B 24.8936,C -2.3815,E1 25.1396,E2 420.9702} C_DIS
LIN {X 67.6628,Y 35.9419,Z 83,A 21.7567,B 24.8942,C -2.3746,E1 25.1419,E2 422.7544} C_DIS
LIN {X 68.9334,Y 33.4405,Z 83,A 19.6617,B 24.8947,C -2.3689,E1 25.1445,E2 424.8517} C_DIS
LIN {X 70.0438,Y 31.0498,Z 83,A 17.8234,B 24.8948,C -2.3674,E1 25.1466,E2 426.6838} C_DIS
LIN {X 71.0736,Y 28.6117,Z 83,A 15.9021,B 24.8952,C -2.3634,E1 25.1487,E2 428.6038} C_DIS
LIN {X 72.0705,Y 25.9984,Z 83,A 13.8677,B 24.8956,C -2.3591,E1 25.1507,E2 430.6371} C_DIS
LIN {X 72.7505,Y 24.033,Z 83,A 12.2329,B 24.8962,C -2.3521,E1 25.1521,E2 432.2792} C_DIS
LIN {X 73.5267,Y 21.5384,Z 83,A 10.3776,B 24.8964,C -2.3492,E1 25.1536,E2 434.1307} C_DIS
LIN {X 74.2603,Y 18.8537,Z 83,A 8.1742,B 24.8973,C -2.3392,E1 25.1552,E2 436.3449} C_DIS
LIN {X 74.9597,Y 15.851,Z 83,A 5.9392,B 24.8978,C -2.3343,E1 25.1566,E2 438.5787} C_DIS
LIN {X 75.4715,Y 13.1982,Z 83,A 3.9758,B 24.8982,C -2.3298,E1 25.1576,E2 440.5413} C_DIS
LIN {X 75.8273,Y 10.9666,Z 83,A 2.1457,B 24.899,C -2.3203,E1 25.1584,E2 442.383} C_DIS
LIN {X 76.1757,Y 8.2046,Z 83,A 0.0768,B 24.8995,C -2.3141,E1 25.159,E2 444.4543} C_DIS
LIN {X 76.4244,Y 5.4198,Z 83,A -1.9988,B 24.9001,C -2.308,E1 25.1595,E2 446.532} C_DIS
LIN {X 76.5777,Y 2.4209,Z 83,A -4.1646,B 24.9005,C -2.3033,E1 25.1597,E2 448.6961} C_DIS
LIN {X 76.6132,Y -0.7219,Z 83,A -6.3961,B 24.9008,C -2.2994,E1 25.1597,E2 450.9234} C_DIS
LIN {X 76.5334,Y -3.5666,Z 83,A -8.4827,B 24.9013,C -2.2939,E1 25.1596,E2 453.0106} C_DIS
LIN {X 76.3936,Y -5.8391,Z 83,A -10.3316,B 24.9021,C -2.284,E1 25.1592,E2 454.8719} C_DIS
LIN {X 76.1202,Y -8.7041,Z 83,A -12.4864,B 24.9027,C -2.2771,E1 25.1586,E2 457.0304} C_DIS
LIN {X 75.7568,Y -11.4445,Z 83,A -14.5264,B 24.9032,C -2.2713,E1 25.1578,E2 459.0719} C_DIS
LIN {X 75.3203,Y -14.038,Z 83,A -16.4025,B 24.9035,C -2.2678,E1 25.1569,E2 460.9453} C_DIS
LIN {X 74.8488,Y -16.3601,Z 83,A -18.1461,B 24.9039,C -2.2631,E1 25.1558,E2 462.6899} C_DIS
LIN {X 74.2578,Y -18.8633,Z 83,A -20.1592,B 24.9047,C -2.2543,E1 25.1545,E2 464.7121} C_DIS
LIN {X 73.3849,Y -22.0162,Z 83,A -22.54,B 24.9051,C -2.2487,E1 25.1527,E2 467.0926} C_DIS
LIN {X 72.6846,Y -24.2285,Z 83,A -24.2977,B 24.9057,C -2.2426,E1 25.1511,E2 468.8547} C_DIS
LIN {X 71.7295,Y -26.9246,Z 83,A -26.4605,B 24.9063,C -2.2353,E1 25.1491,E2 471.0226} C_DIS
LIN {X 70.4904,Y -30.0198,Z 83,A -28.8584,B 24.9067,C -2.2306,E1 25.1465,E2 473.4183} C_DIS
LIN {X 69.5678,Y -32.0996,Z 83,A -30.5863,B 24.9072,C -2.2248,E1 25.1445,E2 475.1507} C_DIS
LIN {X 68.2673,Y -34.7792,Z 83,A -32.7652,B 24.9076,C -2.2197,E1 25.1418,E2 477.33} C_DIS
LIN {X 67.1286,Y -36.9318,Z 83,A -34.5343,B 24.9079,C -2.2159,E1 25.1395,E2 479.0987} C_DIS
LIN {X 65.7311,Y -39.3653,Z 83,A -36.7956,B 24.9088,C -2.205,E1 25.1363,E2 481.3741} C_DIS
LIN {X 64.2264,Y -41.7755,Z 83,A -38.8751,B 24.9092,C -2.2004,E1 25.1331,E2 483.454} C_DIS
LIN {X 62.6297,Y -44.1331,Z 83,A -40.8518,B 24.9092,C -2.1991,E1 25.13,E2 485.424} C_DIS
LIN {X 61.0924,Y -46.2364,Z 83,A -42.9257,B 24.91,C -2.1901,E1 25.1265,E2 487.5092} C_DIS
LIN {X 59.2296,Y -48.6011,Z 83,A -45.1648,B 24.9105,C -2.1846,E1 25.1226,E2 489.7511} C_DIS
LIN {X 57.3278,Y -50.8297,Z 83,A -47.2958,B 24.9108,C -2.1808,E1 25.1187,E2 491.8814} C_DIS
LIN {X 55.2217,Y -53.1091,Z 83,A -49.6073,B 24.9112,C -2.1753,E1 25.1143,E2 494.1957} C_DIS
LIN {X 53.0956,Y -55.2347,Z 83,A -51.8921,B 24.9118,C -2.1689,E1 25.1097,E2 496.4862} C_DIS
LIN {X 50.7498,Y -57.3993,Z 83,A -54.2597,B 24.9122,C -2.1639,E1 25.1048,E2 498.8561} C_DIS
LIN {X 48.3067,Y -59.4683,Z 83,A -56.5465,B 24.9123,C -2.1618,E1 25.0999,E2 501.139} C_DIS
LIN {X 46.2254,Y -61.1006,Z 83,A -58.5482,B 24.9127,C -2.1569,E1 25.0954,E2 503.145} C_DIS
LIN {X 44.1211,Y -62.6383,Z 83,A -60.3047,B 24.9127,C -2.1586,E1 25.0915,E2 504.8914} C_DIS
LIN {X 42.4088,Y -63.8089,Z 83,A -62.0785,B 24.9134,C -2.149,E1 25.0873,E2 506.6819} C_DIS
LIN {X 39.972,Y -65.3627,Z 83,A -64.1503,B 24.9135,C -2.1475,E1 25.0824,E2 508.7505} C_DIS
LIN {X 37.5595,Y -66.7783,Z 83,A -66.3092,B 24.914,C -2.1419,E1 25.0772,E2 510.9164} C_DIS
LIN {X 34.6155,Y -68.3509,Z 83,A -68.7152,B 24.914,C -2.1403,E1 25.0712,E2 513.3194} C_DIS
LIN {X 31.9456,Y -69.6395,Z 83,A -70.7825,B 24.914,C -2.1411,E1 25.066,E2 515.3794} C_DIS
LIN {X 30.0052,Y -70.4966,Z 83,A -72.5494,B 24.9146,C -2.1336,E1 25.0615,E2 517.1598} C_DIS
LIN {X 27.5032,Y -71.5104,Z 83,A -74.6261,B 24.915,C -2.1291,E1 25.0561,E2 519.2425} C_DIS
LIN {X 24.921,Y -72.4511,Z 83,A -76.6919,B 24.9152,C -2.1262,E1 25.0506,E2 521.3111} C_DIS
LIN {X 22.2136,Y -73.3264,Z 83,A -78.826,B 24.9154,C -2.1235,E1 25.0449,E2 523.4476} C_DIS
LIN {X 19.5107,Y -74.0914,Z 83,A -80.7554,B 24.9152,C -2.1261,E1 25.0398,E2 525.3677} C_DIS
LIN {X 17.4957,Y -74.592,Z 83,A -82.382,B 24.9155,C -2.1226,E1 25.0353,E2 527.0005} C_DIS
LIN {X 14.7474,Y -75.1837,Z 83,A -84.4761,B 24.9156,C -2.121,E1 25.0296,E2 529.0957} C_DIS
LIN {X 12.1593,Y -75.6463,Z 83,A -86.3667,B 24.9156,C -2.1216,E1 25.0244,E2 530.9829} C_DIS
LIN {X 9.5561,Y -76.0182,Z 83,A -88.3631,B 24.9158,C -2.1195,E1 25.0189,E2 532.9826} C_DIS
LIN {X 7.2927,Y -76.2685,Z 83,A -90.0999,B 24.9159,C -2.1176,E1 25.014,E2 534.7228} C_DIS
LIN {X 4.6924,Y -76.4735,Z 83,A -91.9808,B 24.9159,C -2.1186,E1 25.0088,E2 536.6003} C_DIS
LIN {X 2.3169,Y -76.5809,Z 83,A -93.8695,B 24.9161,C -2.115,E1 25.0035,E2 538.4972} C_DIS
LIN {X 2.3169,Y -76.5809,Z 83,A -93.8695,B 24.9161,C -2.115,E1 25.0035,E2 538.4972} C_DIS
Enddeposition()
LIN {X 0.567,Y -85.5196,Z 84,A -94.3617,B 24.9257,C -1.9901,E1 25.0013,E2 539.2856} C_DIS
Startdeposition()
$VEL.CP = VEL_PRINT
LIN {X 3.2114,Y -85.4624,Z 84,A -92.2377,B 24.9249,C -2.0018,E1 25.0073,E2 537.1344} C_DIS
LIN {X 5.3078,Y -85.3578,Z 84,A -90.8722,B 24.9249,C -2.0011,E1 25.0111,E2 535.7712} C_DIS
LIN {X 7.401,Y -85.2019,Z 84,A -89.4276,B 24.9248,C -2.003,E1 25.0151,E2 534.3228} C_DIS
LIN {X 9.4265,Y -85.002,Z 84,A -88.0286,B 24.9246,C -2.0049,E1 25.019,E2 532.9203} C_DIS
LIN {X 11.5098,Y -84.745,Z 84,A -86.6244,B 24.9246,C -2.0057,E1 25.0229,E2 531.5152} C_DIS
LIN {X 13.6488,Y -84.4266,Z 84,A -85.2546,B 24.9246,C -2.0042,E1 25.0267,E2 530.1502} C_DIS
LIN {X 15.7166,Y -84.0662,Z 84,A -83.8509,B 24.9246,C -2.0052,E1 25.0305,E2 528.7456} C_DIS
LIN {X 17.7128,Y -83.6687,Z 84,A -82.4498,B 24.9244,C -2.0076,E1 25.0344,E2 527.3406} C_DIS
LIN {X 19.8226,Y -83.1937,Z 84,A -81.0439,B 24.9244,C -2.0076,E1 25.0382,E2 525.9367} C_DIS
LIN {X 21.7969,Y -82.6988,Z 84,A -79.6065,B 24.9241,C -2.0114,E1 25.0421,E2 524.4925} C_DIS
LIN {X 24.2553,Y -82.0098,Z 84,A -77.8034,B 24.9238,C -2.0163,E1 25.047,E2 522.6808} C_DIS
LIN {X 26.8873,Y -81.1862,Z 84,A -76.0945,B 24.9239,C -2.014,E1 25.0515,E2 520.9806} C_DIS
LIN {X 28.8716,Y -80.5019,Z 84,A -74.7318,B 24.9239,C -2.0144,E1 25.0551,E2 519.6198} C_DIS
LIN {X 30.7915,Y -79.7876,Z 84,A -73.2945,B 24.9236,C -2.0183,E1 25.0589,E2 518.1761} C_DIS
LIN {X 32.7283,Y -79.013,Z 84,A -71.7544,B 24.9231,C -2.025,E1 25.0629,E2 516.6237} C_DIS
LIN {X 35.6143,Y -77.7548,Z 84,A -69.7995,B 24.9233,C -2.0231,E1 25.0678,E2 514.6782} C_DIS
LIN {X 37.5118,Y -76.8574,Z 84,A -68.3891,B 24.9231,C -2.0255,E1 25.0714,E2 513.2658} C_DIS
LIN {X 39.5619,Y -75.8214,Z 84,A -67.0168,B 24.9233,C -2.0226,E1 25.0748,E2 511.9043} C_DIS
LIN {X 41.2378,Y -74.9242,Z 84,A -65.5878,B 24.9227,C -2.0299,E1 25.0783,E2 510.4621} C_DIS
LIN {X 43.0641,Y -73.8896,Z 84,A -64.1873,B 24.9226,C -2.0322,E1 25.0817,E2 509.0602} C_DIS
LIN {X 45.4364,Y -72.4533,Z 84,A -62.2779,B 24.9222,C -2.0375,E1 25.0862,E2 507.1445} C_DIS
LIN {X 47.7648,Y -70.9401,Z 84,A -60.6583,B 24.9225,C -2.033,E1 25.09,E2 505.5407} C_DIS
LIN {X 49.2449,Y -69.9224,Z 84,A -59.3236,B 24.922,C -2.0398,E1 25.0931,E2 504.1946} C_DIS
LIN {X 50.946,Y -68.6928,Z 84,A -57.9235,B 24.9218,C -2.0425,E1 25.0962,E2 502.793} C_DIS
LIN {X 52.6664,Y -67.3824,Z 84,A -56.4452,B 24.9215,C -2.0466,E1 25.0995,E2 501.3104} C_DIS
LIN {X 54.3042,Y -66.0696,Z 84,A -55.0821,B 24.9213,C -2.0483,E1 25.1025,E2 499.9487} C_DIS
LIN {X 55.9093,Y -64.717,Z 84,A -53.4892,B 24.9206,C -2.0577,E1 25.1059,E2 498.3396} C_DIS
LIN {X 58.2534,Y -62.6153,Z 84,A -51.6237,B 24.9209,C -2.0544,E1 25.1097,E2 496.4895} C_DIS
LIN {X 59.7725,Y -61.1668,Z 84,A -50.2247,B 24.9206,C -2.0575,E1 25.1125,E2 495.089} C_DIS
LIN {X 61.9398,Y -58.9716,Z 84,A -48.1297,B 24.9202,C -2.0635,E1 25.1166,E2 492.9888} C_DIS
LIN {X 63.3684,Y -57.4338,Z 84,A -46.4793,B 24.9192,C -2.0753,E1 25.1197,E2 491.3177} C_DIS
LIN {X 65.4395,Y -55.0625,Z 84,A -44.5967,B 24.9194,C -2.073,E1 25.1231,E2 489.4491} C_DIS
LIN {X 66.771,Y -53.4399,Z 84,A -43.1985,B 24.9191,C -2.0765,E1 25.1256,E2 488.0493} C_DIS
LIN {X 68.1006,Y -51.7343,Z 84,A -41.6279,B 24.9185,C -2.0845,E1 25.1283,E2 486.4672} C_DIS
LIN {X 69.9224,Y -49.2449,Z 84,A -39.6796,B 24.9184,C -2.0861,E1 25.1314,E2 484.5246} C_DIS
LIN {X 71.1098,Y -47.5141,Z 84,A -38.3062,B 24.9182,C -2.0889,E1 25.1336,E2 483.1514} C_DIS
LIN {X 72.2882,Y -45.7007,Z 84,A -36.9427,B 24.9181,C -2.09,E1 25.1356,E2 481.792} C_DIS
LIN {X 73.388,Y -43.9129,Z 84,A -35.545,B 24.9178,C -2.0937,E1 25.1377,E2 480.3927} C_DIS
LIN {X 74.4435,Y -42.0986,Z 84,A -34.1084,B 24.9174,C -2.0988,E1 25.1397,E2 478.9515} C_DIS
LIN {X 75.7422,Y -39.7123,Z 84,A -32.2057,B 24.9167,C -2.107,E1 25.1422,E2 477.0395} C_DIS
LIN {X 76.885,Y -37.4545,Z 84,A -30.6156,B 24.9167,C -2.1084,E1 25.1442,E2 475.4546} C_DIS
LIN {X 77.7548,Y -35.6143,Z 84,A -29.2606,B 24.9163,C -2.1122,E1 25.1458,E2 474.098} C_DIS
LIN {X 78.6302,Y -33.6368,Z 84,A -27.8608,B 24.9161,C -2.1149,E1 25.1473,E2 472.6995} C_DIS
LIN {X 79.432,Y -31.697,Z 84,A -26.4246,B 24.9157,C -2.1202,E1 25.1488,E2 471.2587} C_DIS
LIN {X 80.5237,Y -28.8119,Z 84,A -24.1849,B 24.9147,C -2.1325,E1 25.151,E2 469.0024} C_DIS
LIN {X 81.5297,Y -25.8285,Z 84,A -22.0647,B 24.9142,C -2.1394,E1 25.1528,E2 466.8778} C_DIS
LIN {X 82.4417,Y -22.7487,Z 84,A -20.1399,B 24.9142,C -2.1383,E1 25.1543,E2 464.9666} C_DIS
LIN {X 82.9601,Y -20.7804,Z 84,A -18.7484,B 24.9138,C -2.1436,E1 25.1553,E2 463.5708} C_DIS
LIN {X 83.4586,Y -18.676,Z 84,A -17.3469,B 24.9136,C -2.1465,E1 25.1562,E2 462.1705} C_DIS
LIN {X 83.8798,Y -16.6847,Z 84,A -15.9574,B 24.9132,C -2.1517,E1 25.1569,E2 460.7767} C_DIS
LIN {X 84.3179,Y -14.2987,Z 84,A -14.4676,B 24.9132,C -2.1523,E1 25.1577,E2 459.2945} C_DIS
LIN {X 84.6064,Y -12.4859,Z 84,A -12.9557,B 24.912,C -2.1659,E1 25.1583,E2 457.7592} C_DIS
LIN {X 85.002,Y -9.4265,Z 84,A -11.1051,B 24.912,C -2.1651,E1 25.1589,E2 455.9216} C_DIS
LIN {X 85.2128,Y -7.2742,Z 84,A -9.7056,B 24.9118,C -2.168,E1 25.1593,E2 454.5234} C_DIS
LIN {X 85.3621,Y -5.2443,Z 84,A -8.3128,B 24.9114,C -2.1734,E1 25.1595,E2 453.1263} C_DIS
LIN {X 85.4651,Y -3.1479,Z 84,A -6.879,B 24.911,C -2.1788,E1 25.1597,E2 451.6881} C_DIS
LIN {X 85.5166,Y -1.0495,Z 84,A -5.2467,B 24.9099,C -2.1911,E1 25.1597,E2 450.0365} C_DIS
LIN {X 85.4954,Y 2.1624,Z 84,A -3.3827,B 24.9102,C -2.1881,E1 25.1597,E2 448.1908} C_DIS
LIN {X 85.4165,Y 4.2599,Z 84,A -1.986,B 24.9099,C -2.1922,E1 25.1595,E2 446.7926} C_DIS
LIN {X 85.2913,Y 6.2915,Z 84,A -0.4245,B 24.9089,C -2.2034,E1 25.1592,E2 445.2141} C_DIS
LIN {X 85.002,Y 9.4265,Z 84,A 1.4996,B 24.9089,C -2.2036,E1 25.1587,E2 443.3007} C_DIS
LIN {X 84.745,Y 11.5098,Z 84,A 2.8961,B 24.9086,C -2.2077,E1 25.1582,E2 441.9028} C_DIS
LIN {X 84.4266,Y 13.6488,Z 84,A 4.2587,B 24.9084,C -2.2093,E1 25.1576,E2 440.5446} C_DIS
LIN {X 84.0662,Y 15.7166,Z 84,A 5.6951,B 24.908,C -2.2147,E1 25.1569,E2 439.1038} C_DIS
LIN {X 83.6552,Y 17.775,Z 84,A 7.0524,B 24.9078,C -2.2173,E1 25.1561,E2 437.7481} C_DIS
LIN {X 83.1937,Y 19.8226,Z 84,A 8.4488,B 24.9074,C -2.2213,E1 25.1552,E2 436.3504} C_DIS
LIN {X 82.6822,Y 21.8583,Z 84,A 9.885,B 24.907,C -2.2266,E1 25.1542,E2 434.91} C_DIS
LIN {X 82.139,Y 23.8199,Z 84,A 11.2397,B 24.9067,C -2.2304,E1 25.1532,E2 433.5541} C_DIS
LIN {X 81.3976,Y 26.2366,Z 84,A 13.0651,B 24.9059,C -2.24,E1 25.1517,E2 431.7164} C_DIS
LIN {X 80.5019,Y 28.8716,Z 84,A 14.7354,B 24.9059,C -2.2388,E1 25.1501,E2 430.0582} C_DIS
LIN {X 79.7924,Y 30.7793,Z 84,A 16.1669,B 24.9054,C -2.2451,E1 25.1487,E2 428.6199} C_DIS
LIN {X 79.013,Y 32.7283,Z 84,A 17.5269,B 24.9052,C -2.2476,E1 25.1473,E2 427.2616} C_DIS
LIN {X 78.186,Y 34.6575,Z 84,A 19.1456,B 24.9043,C -2.2588,E1 25.1454,E2 425.6251} C_DIS
LIN {X 76.8574,Y 37.5118,Z 84,A 21.0206,B 24.9045,C -2.2568,E1 25.1432,E2 423.7651} C_DIS
LIN {X 75.884,Y 39.443,Z 84,A 22.4216,B 24.9043,C -2.2591,E1 25.1414,E2 422.366} C_DIS
LIN {X 74.9242,Y 41.2378,Z 84,A 23.8538,B 24.9037,C -2.2651,E1 25.1395,E2 420.9271} C_DIS
LIN {X 73.8896,Y 43.0641,Z 84,A 25.2519,B 24.9034,C -2.2686,E1 25.1376,E2 419.528} C_DIS
LIN {X 72.7768,Y 44.9185,Z 84,A 26.6155,B 24.9034,C -2.2695,E1 25.1356,E2 418.1691} C_DIS
LIN {X 71.6525,Y 46.691,Z 84,A 28.014,B 24.9031,C -2.2729,E1 25.1335,E2 416.7697} C_DIS
LIN {X 70.2582,Y 48.7618,Z 84,A 29.8477,B 24.9023,C -2.2826,E1 25.1306,E2 414.9222} C_DIS
LIN {X 68.6546,Y 50.9969,Z 84,A 31.5498,B 24.9023,C -2.2823,E1 25.1278,E2 413.2289} C_DIS
LIN {X 67.3824,Y 52.6664,Z 84,A 32.9485,B 24.902,C -2.2855,E1 25.1254,E2 411.8295} C_DIS
LIN {X 66.1102,Y 54.2553,Z 84,A 34.522,B 24.9011,C -2.2957,E1 25.1226,E2 410.239} C_DIS
LIN {X 64.026,Y 56.6992,Z 84,A 36.4463,B 24.9014,C -2.293,E1 25.1191,E2 408.3299} C_DIS
LIN {X 62.5452,Y 58.3279,Z 84,A 37.8106,B 24.9014,C -2.2926,E1 25.1165,E2 406.9725} C_DIS
LIN {X 61.1668,Y 59.7725,Z 84,A 39.2452,B 24.9009,C -2.2987,E1 25.1137,E2 405.5296} C_DIS
LIN {X 59.7273,Y 61.2115,Z 84,A 40.6396,B 24.9005,C -2.3026,E1 25.1109,E2 404.1319} C_DIS
LIN {X 58.1602,Y 62.7019,Z 84,A 42.2317,B 24.8999,C -2.3103,E1 25.1077,E2 402.5281} C_DIS
LIN {X 55.8613,Y 64.7588,Z 84,A 44.1028,B 24.9001,C -2.3078,E1 25.1038,E2 400.6702} C_DIS
LIN {X 54.2058,Y 66.1503,Z 84,A 45.5457,B 24.8999,C -2.3104,E1 25.1007,E2 399.2268} C_DIS
LIN {X 52.5661,Y 67.4606,Z 84,A 46.9065,B 24.8998,C -2.3114,E1 25.0977,E2 397.8685} C_DIS
LIN {X 50.8947,Y 68.7304,Z 84,A 48.535,B 24.8989,C -2.3212,E1 25.094,E2 396.2228} C_DIS
LIN {X 48.3831,Y 70.5214,Z 84,A 50.6336,B 24.8985,C -2.3257,E1 25.0892,E2 394.1208} C_DIS
LIN {X 45.7007,Y 72.2882,Z 84,A 52.511,B 24.899,C -2.3201,E1 25.0848,E2 392.2628} C_DIS
LIN {X 43.8046,Y 73.4519,Z 84,A 53.9186,B 24.899,C -2.3196,E1 25.0815,E2 390.8606} C_DIS
LIN {X 41.5915,Y 74.7267,Z 84,A 55.8123,B 24.8983,C -2.328,E1 25.0769,E2 388.9529} C_DIS
LIN {X 39.33,Y 75.9426,Z 84,A 57.4179,B 24.8984,C -2.3265,E1 25.0729,E2 387.3552} C_DIS
LIN {X 37.4545,Y 76.885,Z 84,A 58.8597,B 24.8982,C -2.3294,E1 25.0693,E2 385.9105} C_DIS
LIN {X 35.401,Y 77.851,Z 84,A 60.3626,B 24.8981,C -2.3306,E1 25.0655,E2 384.4086} C_DIS
LIN {X 33.6368,Y 78.6301,Z 84,A 61.8449,B 24.8974,C -2.3381,E1 25.0617,E2 382.9121} C_DIS
LIN {X 30.7198,Y 79.8149,Z 84,A 63.7304,B 24.8979,C -2.333,E1 25.0568,E2 381.0427} C_DIS
LIN {X 28.7518,Y 80.5448,Z 84,A 65.1735,B 24.8977,C -2.3355,E1 25.053,E2 379.5968} C_DIS
LIN {X 26.7551,Y 81.2298,Z 84,A 66.5789,B 24.8976,C -2.3364,E1 25.0493,E2 378.192} C_DIS
LIN {X 24.765,Y 81.8586,Z 84,A 67.9414,B 24.8976,C -2.3364,E1 25.0457,E2 376.8322} C_DIS
LIN {X 22.8101,Y 82.4251,Z 84,A 69.3797,B 24.8973,C -2.3396,E1 25.0418,E2 375.3884} C_DIS
LIN {X 20.3243,Y 83.0713,Z 84,A 71.1899,B 24.897,C -2.3434,E1 25.0369,E2 373.5719} C_DIS
LIN {X 17.7128,Y 83.6687,Z 84,A 72.8542,B 24.8972,C -2.3402,E1 25.0324,E2 371.9174} C_DIS
LIN {X 15.5915,Y 84.0895,Z 84,A 74.2617,B 24.8973,C -2.3395,E1 25.0285,E2 370.5132} C_DIS
LIN {X 13.5232,Y 84.4468,Z 84,A 75.9311,B 24.8965,C -2.3482,E1 25.0239,E2 368.825} C_DIS
LIN {X 10.4057,Y 84.8873,Z 84,A 77.9195,B 24.8968,C -2.3449,E1 25.0184,E2 366.846} C_DIS
LIN {X 7.2742,Y 85.2128,Z 84,A 79.8844,B 24.8972,C -2.3407,E1 25.013,E2 364.8923} C_DIS
LIN {X 5.0155,Y 85.3748,Z 84,A 81.2976,B 24.8975,C -2.3375,E1 25.009,E2 363.4873} C_DIS
LIN {X 3.1479,Y 85.4651,Z 84,A 82.7312,B 24.897,C -2.343,E1 25.005,E2 362.0411} C_DIS
LIN {X 1.0495,Y 85.5166,Z 84,A 84.296,B 24.8966,C -2.3476,E1 25.0006,E2 360.4654} C_DIS
LIN {X -2.0988,Y 85.4973,Z 84,A 86.2485,B 24.8971,C -2.3423,E1 24.9952,E2 358.5254} C_DIS
LIN {X -4.2599,Y 85.4165,Z 84,A 87.6612,B 24.8971,C -2.3407,E1 24.9913,E2 357.1162} C_DIS
LIN {X -6.2915,Y 85.2913,Z 84,A 89.063,B 24.8971,C -2.3413,E1 24.9873,E2 355.7124} C_DIS
LIN {X -8.446,Y 85.1046,Z 84,A 90.6894,B 24.8967,C -2.346,E1 24.9828,E2 354.074} C_DIS
LIN {X -11.5098,Y 84.745,Z 84,A 92.7133,B 24.897,C -2.3435,E1 24.9772,E2 352.0547} C_DIS
LIN {X -14.6212,Y 84.264,Z 84,A 94.6959,B 24.8974,C -2.3382,E1 24.9718,E2 350.0829} C_DIS
LIN {X -16.6847,Y 83.8798,Z 84,A 96.0668,B 24.8976,C -2.336,E1 24.968,E2 348.7157} C_DIS
LIN {X -19.1253,Y 83.3556,Z 84,A 97.899,B 24.8973,C -2.3393,E1 24.963,E2 346.8732} C_DIS
LIN {X -21.7969,Y 82.6988,Z 84,A 99.6274,B 24.8978,C -2.3341,E1 24.9583,E2 345.1548} C_DIS
LIN {X -23.8199,Y 82.139,Z 84,A 101.0371,B 24.8979,C -2.3327,E1 24.9546,E2 343.7462} C_DIS
LIN {X -25.8285,Y 81.5297,Z 84,A 102.6341,B 24.8975,C -2.3368,E1 24.9503,E2 342.1367} C_DIS
LIN {X -28.8716,Y 80.5019,Z 84,A 104.5272,B 24.8984,C -2.3265,E1 24.9453,E2 340.2644} C_DIS
LIN {X -30.7793,Y 79.7924,Z 84,A 105.9723,B 24.8984,C -2.3271,E1 24.9415,E2 338.8149} C_DIS
LIN {X -32.7283,Y 79.013,Z 84,A 107.3827,B 24.8986,C -2.3252,E1 24.9379,E2 337.4057} C_DIS
LIN {X -34.6575,Y 78.186,Z 84,A 108.7557,B 24.8988,C -2.3222,E1 24.9344,E2 336.0366} C_DIS
LIN {X -36.5658,Y 77.3119,Z 84,A 110.2049,B 24.8988,C -2.3213,E1 24.9307,E2 334.5859} C_DIS
LIN {X -38.5088,Y 76.3623,Z 84,A 111.581,B 24.8993,C -2.3169,E1 24.9273,E2 333.2167} C_DIS
LIN {X -40.3153,Y 75.4246,Z 84,A 112.9894,B 24.8993,C -2.316,E1 24.9238,E2 331.8066} C_DIS
LIN {X -42.2093,Y 74.3808,Z 84,A 114.4044,B 24.8997,C -2.3125,E1 24.9204,E2 330.3958} C_DIS
LIN {X -44.022,Y 73.3225,Z 84,A 115.8159,B 24.8999,C -2.3101,E1 24.917,E2 328.9857} C_DIS
LIN {X -45.8082,Y 72.2201,Z 84,A 117.2283,B 24.9001,C -2.3077,E1 24.9136,E2 327.5746} C_DIS
LIN {X -47.6482,Y 71.0191,Z 84,A 118.6889,B 24.9004,C -2.3045,E1 24.9103,E2 326.1167} C_DIS
LIN {X -49.2449,Y 69.9224,Z 84,A 120.0497,B 24.9004,C -2.3038,E1 24.9071,E2 324.7531} C_DIS
LIN {X -51.7852,Y 68.0624,Z 84,A 122.2065,B 24.9007,C -2.3008,E1 24.9023,E2 322.5958} C_DIS
LIN {X -53.4399,Y 66.771,Z 84,A 123.6193,B 24.9009,C -2.298,E1 24.8992,E2 321.1844} C_DIS
LIN {X -55.1109,Y 65.3982,Z 84,A 125.1186,B 24.9011,C -2.2962,E1 24.896,E2 319.6835} C_DIS
LIN {X -56.6992,Y 64.026,Z 84,A 126.451,B 24.9015,C -2.291,E1 24.8932,E2 318.3584} C_DIS
LIN {X -58.2071,Y 62.6588,Z 84,A 127.8216,B 24.9018,C -2.288,E1 24.8904,E2 316.9893} C_DIS
LIN {X -59.7273,Y 61.2115,Z 84,A 129.2353,B 24.902,C -2.2849,E1 24.8875,E2 315.5771} C_DIS
LIN {X -61.2557,Y 59.6815,Z 84,A 130.652,B 24.9024,C -2.2805,E1 24.8848,E2 314.1648} C_DIS
LIN {X -62.6588,Y 58.2071,Z 84,A 132.0631,B 24.9026,C -2.2785,E1 24.8821,E2 312.7524} C_DIS
LIN {X -64.2025,Y 56.4984,Z 84,A 133.4862,B 24.9032,C -2.2713,E1 24.8794,E2 311.3401} C_DIS
LIN {X -65.4395,Y 55.0625,Z 84,A 135.1396,B 24.9026,C -2.2789,E1 24.8764,E2 309.6612} C_DIS
LIN {X -67.4606,Y 52.5661,Z 84,A 137.0159,B 24.9037,C -2.2655,E1 24.8732,E2 307.808} C_DIS
LIN {X -68.7304,Y 50.8947,Z 84,A 138.4304,B 24.904,C -2.262,E1 24.8708,E2 306.3951} C_DIS
LIN {X -69.9912,Y 49.1459,Z 84,A 140.0402,B 24.904,C -2.2627,E1 24.8682,E2 304.7757} C_DIS
LIN {X -71.6876,Y 46.6379,Z 84,A 142.0025,B 24.9046,C -2.2552,E1 24.8652,E2 302.8214} C_DIS
LIN {X -72.8105,Y 44.8645,Z 84,A 143.4172,B 24.9049,C -2.2515,E1 24.8631,E2 301.4084} C_DIS
LIN {X -73.9213,Y 43.009,Z 84,A 144.8377,B 24.9053,C -2.2466,E1 24.8611,E2 299.9922} C_DIS
LIN {X -74.9242,Y 41.2378,Z 84,A 146.2479,B 24.9055,C -2.2439,E1 24.8592,E2 298.5809} C_DIS
LIN {X -75.9426,Y 39.33,Z 84,A 147.6681,B 24.906,C -2.2389,E1 24.8573,E2 297.1651} C_DIS
LIN {X -76.8574,Y 37.5118,Z 84,A 149.0785,B 24.9062,C -2.2362,E1 24.8556,E2 295.7537} C_DIS
LIN {X -77.781,Y 35.5563,Z 84,A 150.4991,B 24.9066,C -2.2311,E1 24.8539,E2 294.3374} C_DIS
LIN {X -78.6302,Y 33.6368,Z 84,A 151.8751,B 24.907,C -2.2261,E1 24.8524,E2 292.9659} C_DIS
LIN {X -79.432,Y 31.697,Z 84,A 153.3308,B 24.9073,C -2.2232,E1 24.8509,E2 291.509} C_DIS
LIN {X -80.1641,Y 29.7978,Z 84,A 154.7412,B 24.9075,C -2.2203,E1 24.8495,E2 290.0975} C_DIS
LIN {X -81.0811,Y 27.1991,Z 84,A 156.6297,B 24.9079,C -2.2158,E1 24.8477,E2 288.2089} C_DIS
LIN {X -81.8586,Y 24.765,Z 84,A 158.2465,B 24.9086,C -2.2078,E1 24.8464,E2 286.6019} C_DIS
LIN {X -82.4417,Y 22.7487,Z 84,A 159.7023,B 24.9088,C -2.2048,E1 24.8453,E2 285.1449} C_DIS
LIN {X -82.9601,Y 20.7804,Z 84,A 161.1133,B 24.9091,C -2.2018,E1 24.8443,E2 283.7328} C_DIS
LIN {X -83.4586,Y 18.676,Z 84,A 162.5344,B 24.9095,C -2.1965,E1 24.8434,E2 282.316} C_DIS
LIN {X -83.8798,Y 16.6847,Z 84,A 163.9737,B 24.9097,C -2.1943,E1 24.8426,E2 280.8736} C_DIS
LIN {X -84.264,Y 14.6212,Z 84,A 165.324,B 24.9102,C -2.1883,E1 24.842,E2 279.5295} C_DIS
LIN {X -84.6064,Y 12.4858,Z 84,A 166.9814,B 24.9101,C -2.1895,E1 24.8413,E2 277.8595} C_DIS
LIN {X -85.002,Y 9.4265,Z 84,A 168.8647,B 24.911,C -2.1778,E1 24.8407,E2 275.9929} C_DIS
LIN {X -85.2128,Y 7.2742,Z 84,A 170.2841,B 24.9115,C -2.1723,E1 24.8403,E2 274.5779} C_DIS
LIN {X -85.3621,Y 5.2443,Z 84,A 171.9475,B 24.9112,C -2.1763,E1 24.84,E2 272.8951} C_DIS
LIN {X -85.4985,Y 2.0352,Z 84,A 173.9821,B 24.912,C -2.1662,E1 24.8398,E2 270.8724} C_DIS
LIN {X -85.5166,Y -1.0495,Z 84,A 175.9835,B 24.9127,C -2.1578,E1 24.8398,E2 268.879} C_DIS
LIN {X -85.4444,Y -3.6302,Z 84,A 177.8464,B 24.9128,C -2.156,E1 24.84,E2 267.009} C_DIS
LIN {X -85.2397,Y -6.9377,Z 84,A -179.9711,B 24.9135,C -2.1479,E1 24.8404,E2 264.8328} C_DIS
LIN {X -85.002,Y -9.4265,Z 84,A -178.3519,B 24.914,C -2.1411,E1 24.8409,E2 263.2202} C_DIS
LIN {X -84.745,Y -11.5098,Z 84,A -176.9359,B 24.9144,C -2.1369,E1 24.8414,E2 261.8056} C_DIS
LIN {X -84.4266,Y -13.6488,Z 84,A -175.5545,B 24.9149,C -2.1306,E1 24.842,E2 260.4312} C_DIS
LIN {X -84.0662,Y -15.7166,Z 84,A -174.1386,B 24.9152,C -2.1265,E1 24.8427,E2 259.0166} C_DIS
LIN {X -83.6687,Y -17.7128,Z 84,A -172.5378,B 24.915,C -2.1289,E1 24.8436,E2 257.4007} C_DIS
LIN {X -82.9601,Y -20.7804,Z 84,A -170.6019,B 24.9159,C -2.1176,E1 24.8449,E2 255.4804} C_DIS
LIN {X -82.4077,Y -22.8713,Z 84,A -169.0198,B 24.9159,C -2.1169,E1 24.846,E2 253.8906} C_DIS
LIN {X -81.5297,Y -25.8285,Z 84,A -167.0251,B 24.9166,C -2.1088,E1 24.8477,E2 251.9039} C_DIS
LIN {X -80.8502,Y -27.8816,Z 84,A -165.6044,B 24.917,C -2.1037,E1 24.8489,E2 250.4873} C_DIS
LIN {X -80.1641,Y -29.7978,Z 84,A -164.232,B 24.9173,C -2.1,E1 24.8502,E2 249.116} C_DIS
LIN {X -79.3847,Y -31.8151,Z 84,A -162.7007,B 24.9174,C -2.0981,E1 24.8518,E2 247.5806} C_DIS
LIN {X -78.58,Y -33.7537,Z 84,A -161.1394,B 24.9174,C -2.0985,E1 24.8535,E2 246.0097} C_DIS
LIN {X -77.3119,Y -36.5658,Z 84,A -159.2787,B 24.9183,C -2.0868,E1 24.8557,E2 244.1666} C_DIS
LIN {X -76.3623,Y -38.5088,Z 84,A -157.8608,B 24.9187,C -2.082,E1 24.8574,E2 242.7527} C_DIS
LIN {X -75.4246,Y -40.3153,Z 84,A -156.4494,B 24.9189,C -2.0796,E1 24.8593,E2 241.3394} C_DIS
LIN {X -74.3808,Y -42.2093,Z 84,A -154.9719,B 24.9191,C -2.0766,E1 24.8613,E2 239.8615} C_DIS
LIN {X -73.3225,Y -44.022,Z 84,A -153.6172,B 24.9195,C -2.0714,E1 24.8632,E2 238.5121} C_DIS
LIN {X -72.2545,Y -45.7546,Z 84,A -152.0079,B 24.9193,C -2.0749,E1 24.8656,E2 236.8863} C_DIS
LIN {X -70.5214,Y -48.3831,Z 84,A -150.0846,B 24.9201,C -2.0642,E1 24.8686,E2 234.9788} C_DIS
LIN {X -69.3128,Y -50.0992,Z 84,A -148.6707,B 24.9203,C -2.061,E1 24.8709,E2 233.5657} C_DIS
LIN {X -68.0624,Y -51.7852,Z 84,A -147.2192,B 24.9205,C -2.0589,E1 24.8733,E2 232.1123} C_DIS
LIN {X -66.771,Y -53.4399,Z 84,A -145.8057,B 24.9207,C -2.0558,E1 24.8758,E2 230.6995} C_DIS
LIN {X -65.3056,Y -55.2196,Z 84,A -144.374,B 24.9213,C -2.049,E1 24.8783,E2 229.2775} C_DIS
LIN {X -63.8061,Y -56.9449,Z 84,A -142.5934,B 24.921,C -2.0527,E1 24.8816,E2 227.4799} C_DIS
LIN {X -61.8636,Y -59.0507,Z 84,A -140.8502,B 24.9217,C -2.0434,E1 24.8849,E2 225.7512} C_DIS
LIN {X -60.4739,Y -60.4739,Z 84,A -139.4465,B 24.9217,C -2.0427,E1 24.8877,E2 224.3433} C_DIS
LIN {X -58.9716,Y -61.9398,Z 84,A -138.0713,B 24.922,C -2.0389,E1 24.8905,E2 222.9715} C_DIS
LIN {X -57.4338,Y -63.3684,Z 84,A -136.5135,B 24.922,C -2.0405,E1 24.8937,E2 221.4035} C_DIS
LIN {X -55.0625,Y -65.4395,Z 84,A -134.5031,B 24.9225,C -2.0336,E1 24.8979,E2 219.4017} C_DIS
LIN {X -53.0422,Y -67.0854,Z 84,A -132.6379,B 24.9225,C -2.034,E1 24.902,E2 217.5288} C_DIS
LIN {X -50.5179,Y -69.0063,Z 84,A -130.5466,B 24.9228,C -2.0293,E1 24.9067,E2 215.4411} C_DIS
LIN {X -48.3831,Y -70.5214,Z 84,A -128.894,B 24.9232,C -2.0234,E1 24.9105,E2 213.7969} C_DIS
LIN {X -46.5843,Y -71.7219,Z 84,A -127.4397,B 24.9234,C -2.0213,E1 24.9138,E2 212.3429} C_DIS
LIN {X -44.8645,Y -72.8105,Z 84,A -126.0344,B 24.9234,C -2.0205,E1 24.9172,E2 210.9351} C_DIS
LIN {X -43.0641,Y -73.8896,Z 84,A -124.6239,B 24.9236,C -2.0186,E1 24.9206,E2 209.5247} C_DIS
LIN {X -41.1819,Y -74.9545,Z 84,A -123.2078,B 24.9238,C -2.0157,E1 24.924,E2 208.1115} C_DIS
LIN {X -39.3867,Y -75.9137,Z 84,A -121.8032,B 24.9238,C -2.0151,E1 24.9275,E2 206.7042} C_DIS
LIN {X -36.5081,Y -77.3388,Z 84,A -119.7224,B 24.9242,C -2.0105,E1 24.9327,E2 204.6293} C_DIS
LIN {X -34.4454,Y -78.2785,Z 84,A -118.2582,B 24.9245,C -2.0072,E1 24.9364,E2 203.1693} C_DIS
LIN {X -32.7283,Y -79.013,Z 84,A -116.8689,B 24.9242,C -2.01,E1 24.94,E2 201.77} C_DIS
LIN {X -30.7198,Y -79.8149,Z 84,A -115.4421,B 24.9244,C -2.008,E1 24.9437,E2 200.3449} C_DIS
LIN {X -28.7641,Y -80.5405,Z 84,A -114.0857,B 24.9246,C -2.0055,E1 24.9473,E2 198.9917} C_DIS
LIN {X -26.7665,Y -81.2262,Z 84,A -112.6766,B 24.9246,C -2.0042,E1 24.951,E2 197.583} C_DIS
LIN {X -24.765,Y -81.8586,Z 84,A -111.0581,B 24.9243,C -2.0097,E1 24.9554,E2 195.9488} C_DIS
LIN {X -21.7353,Y -82.7146,Z 84,A -109.1555,B 24.9248,C -2.002,E1 24.9605,E2 194.0615} C_DIS
LIN {X -19.6988,Y -83.2231,Z 84,A -107.7079,B 24.9248,C -2.0025,E1 24.9644,E2 192.6106} C_DIS
LIN {X -17.6505,Y -83.6815,Z 84,A -106.3399,B 24.9249,C -2.0007,E1 24.9681,E2 191.2452} C_DIS
LIN {X -15.5915,Y -84.0895,Z 84,A -104.9328,B 24.9249,C -2.0002,E1 24.972,E2 189.8378} C_DIS
LIN {X -13.586,Y -84.4371,Z 84,A -103.4912,B 24.9249,C -2.0022,E1 24.976,E2 188.3901} C_DIS
LIN {X -11.5098,Y -84.745,Z 84,A -102.0843,B 24.9249,C -2.002,E1 24.9799,E2 186.9827} C_DIS
LIN {X -9.4265,Y -85.002,Z 84,A -100.6171,B 24.9247,C -2.0037,E1 24.9839,E2 185.5104} C_DIS
LIN {X -7.2742,Y -85.2128,Z 84,A -99.2246,B 24.9249,C -2.0018,E1 24.9878,E2 184.1216} C_DIS
LIN {X -5.2443,Y -85.3621,Z 84,A -97.9026,B 24.9249,C -2.0005,E1 24.9915,E2 182.8022} C_DIS
LIN {X -2.8677,Y -85.4737,Z 84,A -96.4335,B 24.9252,C -1.9968,E1 24.9956,E2 181.3417} C_DIS
LIN {X -1.0495,Y -85.5166,Z 84,A -95.0533,B 24.9248,C -2.0021,E1 24.9994,E2 179.9489} C_DIS
LIN {X -1.0495,Y -85.5166,Z 84,A -95.0533,B 24.9248,C -2.0021,E1 24.9994,E2 179.9489} C_DIS
Enddeposition()
LIN {X 0.5554,Y -84.5445,Z 84,A -94.0915,B 24.9238,C -2.0157,E1 25.0022,E2 178.9549} C_DIS
Startdeposition()
$VEL.CP = VEL_PRINT
LIN {X -2.5354,Y -84.5473,Z 84,A -97.9575,B 24.9279,C -1.9605,E1 24.9911,E2 182.9522} C_DIS
LIN {X -7.2904,Y -84.272,Z 84,A -100.2801,B 24.9259,C -1.9877,E1 24.9848,E2 185.2111} C_DIS
LIN {X -10.8245,Y -83.8899,Z 84,A -102.6621,B 24.9259,C -1.9889,E1 24.9782,E2 187.5919} C_DIS
LIN {X -14.1736,Y -83.3897,Z 84,A -104.8836,B 24.9256,C -1.9917,E1 24.9721,E2 189.8088} C_DIS
LIN {X -17.4537,Y -82.7662,Z 84,A -106.986,B 24.9252,C -1.9974,E1 24.9663,E2 191.9001} C_DIS
LIN {X -20.1141,Y -82.159,Z 84,A -109.0499,B 24.9256,C -1.9919,E1 24.9607,E2 193.9799} C_DIS
LIN {X -22.7536,Y -81.4681,Z 84,A -110.8608,B 24.9254,C -1.9941,E1 24.9558,E2 195.7882} C_DIS
LIN {X -25.7814,Y -80.561,Z 84,A -113.1032,B 24.9255,C -1.9927,E1 24.9498,E2 198.0379} C_DIS
LIN {X -29.4425,Y -79.2972,Z 84,A -115.6909,B 24.9253,C -1.996,E1 24.943,E2 200.6229} C_DIS
LIN {X -32.5428,Y -78.0753,Z 84,A -118.5432,B 24.9264,C -1.9809,E1 24.9355,E2 203.5175} C_DIS
LIN {X -35.8274,Y -76.6231,Z 84,A -120.0139,B 24.9241,C -2.0116,E1 24.932,E2 204.9187} C_DIS
LIN {X -37.5571,Y -75.7901,Z 84,A -121.554,B 24.9245,C -2.0062,E1 24.9281,E2 206.4758} C_DIS
LIN {X -39.5253,Y -74.7827,Z 84,A -123.1657,B 24.9246,C -2.0048,E1 24.9241,E2 208.0952} C_DIS
LIN {X -42.5583,Y -73.1006,Z 84,A -125.5861,B 24.9246,C -2.0059,E1 24.9182,E2 210.52} C_DIS
LIN {X -45.4774,Y -71.3201,Z 84,A -127.6548,B 24.9238,C -2.0165,E1 24.9133,E2 212.57} C_DIS
LIN {X -47.8913,Y -69.7232,Z 84,A -129.9032,B 24.9241,C -2.0114,E1 24.9081,E2 214.8382} C_DIS
LIN {X -50.1246,Y -68.134,Z 84,A -131.7281,B 24.9238,C -2.0154,E1 24.9039,E2 216.6597} C_DIS
LIN {X -53.1392,Y -65.8098,Z 84,A -134.2002,B 24.9233,C -2.0231,E1 24.8985,E2 219.1228} C_DIS
LIN {X -55.7588,Y -63.6055,Z 84,A -136.5929,B 24.9231,C -2.0254,E1 24.8935,E2 221.5191} C_DIS
LIN {X -58.0587,Y -61.5133,Z 84,A -138.8403,B 24.9231,C -2.0257,E1 24.8888,E2 223.7751} C_DIS
LIN {X -60.0936,Y -59.5269,Z 84,A -140.5905,B 24.9224,C -2.0346,E1 24.8854,E2 225.5114} C_DIS
LIN {X -62.3617,Y -57.1462,Z 84,A -142.8724,B 24.9221,C -2.038,E1 24.881,E2 227.7953} C_DIS
LIN {X -64.7902,Y -54.379,Z 84,A -145.3451,B 24.9216,C -2.0442,E1 24.8765,E2 230.2643} C_DIS
LIN {X -66.5526,Y -52.2065,Z 84,A -147.2348,B 24.9213,C -2.0488,E1 24.8733,E2 232.152} C_DIS
LIN {X -68.3058,Y -49.8899,Z 84,A -149.1567,B 24.9208,C -2.0549,E1 24.8701,E2 234.0686} C_DIS
LIN {X -70.4538,Y -46.8085,Z 84,A -151.497,B 24.9199,C -2.0669,E1 24.8664,E2 236.3919} C_DIS
LIN {X -71.9623,Y -44.4553,Z 84,A -153.8851,B 24.9206,C -2.0581,E1 24.8628,E2 238.813} C_DIS
LIN {X -74.759,Y -39.5702,Z 84,A -157.2382,B 24.9188,C -2.081,E1 24.8583,E2 242.1292} C_DIS
LIN {X -75.8794,Y -37.377,Z 84,A -159.2648,B 24.9192,C -2.0757,E1 24.8557,E2 244.1793} C_DIS
LIN {X -77.2941,Y -34.358,Z 84,A -161.525,B 24.9187,C -2.082,E1 24.853,E2 246.4369} C_DIS
LIN {X -78.2117,Y -32.2138,Z 84,A -163.1719,B 24.9185,C -2.0847,E1 24.8513,E2 248.0864} C_DIS
LIN {X -79.246,Y -29.5788,Z 84,A -164.8463,B 24.9175,C -2.0968,E1 24.8496,E2 249.7412} C_DIS
LIN {X -80.1546,Y -27.017,Z 84,A -167.0773,B 24.9179,C -2.0917,E1 24.8476,E2 251.9972} C_DIS
Enddeposition()
END
